(* IEC 61131-3 sources: Elmo_Master/Lasal_PRG/Elmo_EtherCAT_Test_4Axis/Class/LMCControlCommandService (part 3) *)

		groupHeaderPublished := FALSE;
		if restorePreempt & restoredGroupActive then
			// The compact suffix is shared. Restore the complete captured suffix
			// even when the active Group is disjoint from the selected rollback
			// axes, and keep its shared header invalid until every record is done.
			identityHeaderBase := LMC_OWNER_IDENTITY_GROUP_HEADER_BASE;
			OwnershipIdentityState[identityHeaderBase] := 0;
			_memcpy(ptr1:=#OwnershipIdentityState[0],
				ptr2:=#OwnershipPreemptedIdentityState[0],
				cntr:=LMC_OWNER_IDENTITY_SUFFIX_BYTES);
			_memset(dest:=#OwnershipIdentityState[identityHeaderBase],
				usByte:=0, cntr:=40);
			OwnershipIdentityState[identityHeaderBase + 1] :=
				LMC_OWNER_IDENTITY_VERSION;
			OwnershipIdentityState[identityHeaderBase + 2]$UDINT :=
				restoredGroupIdentitySize;
			OwnershipIdentityState[identityHeaderBase + 3]$UDINT :=
				restoredGroupToken;
			OwnershipIdentityState[identityHeaderBase + 4]$UDINT :=
				restoredGroupGeneration;
			OwnershipIdentityState[identityHeaderBase + 5]$UDINT :=
				restoredGroupMask;
			OwnershipIdentityState[identityHeaderBase + 6]$UDINT :=
				restoredGroupSession;
			OwnershipIdentityState[identityHeaderBase + 7]$UDINT :=
				restoredGroupSequence;
			OwnershipIdentityState[identityHeaderBase + 8]$UDINT :=
				TO_UDINT(restoredGroupCommand) or
				(TO_UDINT(restoredGroupReference) shl 16);
			OwnershipIdentityState[identityHeaderBase + 9]$UDINT :=
				TO_UDINT(LMC_OWNER_KIND_GROUP) or
				(TO_UDINT(LMC_OWNER_RESOURCE_AXIS) shl 8) or
				(TO_UDINT(restoredGroupAdmissionMode) shl 16);
			groupHeaderPublished := TRUE;
		end_if;
		axisIndex := 1;
		while axisIndex <= LMC_OWNER_AXIS_COUNT do
			case axisIndex of
				1: axisBit := 0x00000001;
				2: axisBit := 0x00000002;
				3: axisBit := 0x00000004;
				4: axisBit := 0x00000008;
				5: axisBit := 0x00000010;
				6: axisBit := 0x00000020;
				7: axisBit := 0x00000040;
				8: axisBit := 0x00000080;
				9: axisBit := 0x00000100;
			else
				axisBit := 0;
			end_case;
			if (expectedAxisMask and axisBit) <> 0 then
				recordBase := LMC_OWNER_GLOBAL_SLOTS +
					((axisIndex - 1) * LMC_OWNER_AXIS_STRIDE);
				clearIndex := (axisIndex - 1) * LMC_OWNER_AXIS_STRIDE;
				observerBase := (axisIndex - 1) *
					LMC_OWNER_OBSERVER_STRIDE;
				identityHeaderBase := LMC_OWNER_IDENTITY_AXIS_HEADER_BASE +
					((axisIndex - 1) *
					 LMC_OWNER_IDENTITY_AXIS_HEADER_STRIDE);
				OwnershipIdentityState[identityHeaderBase] := 0;
				_memset(dest:=#OwnershipIdentityState[identityHeaderBase],
					usByte:=0,
					cntr:=LMC_OWNER_IDENTITY_AXIS_HEADER_STRIDE * 4);
				if restorePreempt then
					_memcpy(ptr1:=#OwnershipState[recordBase],
						ptr2:=#OwnershipPreemptedState[clearIndex],
						cntr:=LMC_OWNER_AXIS_STRIDE * 4);
					_memcpy(ptr1:=#OwnershipObserverState[observerBase],
						ptr2:=#OwnershipPreemptedIdentityState[
						 LMC_OWNER_PREEMPT_OBSERVER_BASE + observerBase],
						cntr:=LMC_OWNER_OBSERVER_STRIDE * 4);
				else
					_memcpy(ptr1:=#OwnershipState[recordBase],
						ptr2:=#OwnershipLeaseState[clearIndex],
						cntr:=LMC_OWNER_AXIS_STRIDE * 4);
					_memset(dest:=#OwnershipObserverState[observerBase],
						usByte:=0, cntr:=LMC_OWNER_OBSERVER_STRIDE * 4);
				end_if;
				if OwnershipState[recordBase + 1] <> LMC_OWNER_STATE_IDLE then
				identitySize := OwnershipState[recordBase + 15]$UDINT;
				identityTailSize := 0;
				if identitySize > LMC_OWNER_IDENTITY_PREFIX_BYTES then
					identityTailSize := identitySize -
						LMC_OWNER_IDENTITY_PREFIX_BYTES;
				end_if;
				identityPackedCommand :=
					TO_UDINT(OwnershipState[recordBase + 3]) or
					(TO_UDINT(OwnershipState[recordBase + 12]) shl 16);
				identityPackedOwner :=
					TO_UDINT(OwnershipState[recordBase + 2]) or
					(TO_UDINT(OwnershipState[recordBase + 13]) shl 8) or
					(TO_UDINT(OwnershipState[recordBase + 14]) shl 16);
				if OwnershipState[recordBase + 2] =
				   LMC_OWNER_KIND_GROUP then
					if groupHeaderPublished = FALSE then
						identityHeaderBase :=
							LMC_OWNER_IDENTITY_GROUP_HEADER_BASE;
						OwnershipIdentityState[identityHeaderBase] := 0;
						if restorePreempt then
							_memcpy(ptr1:=#OwnershipIdentityState[0],
								ptr2:=#OwnershipPreemptedIdentityState[0],
								cntr:=LMC_OWNER_IDENTITY_SUFFIX_BYTES);
							_memset(dest:=#OwnershipIdentityState[
								identityHeaderBase], usByte:=0, cntr:=40);
							OwnershipIdentityState[identityHeaderBase + 1] :=
								LMC_OWNER_IDENTITY_VERSION;
							OwnershipIdentityState[identityHeaderBase + 2]$UDINT :=
								identitySize;
							OwnershipIdentityState[identityHeaderBase + 3]$UDINT :=
								OwnershipState[recordBase + 4]$UDINT;
							OwnershipIdentityState[identityHeaderBase + 4]$UDINT :=
								OwnershipState[recordBase + 5]$UDINT;
							OwnershipIdentityState[identityHeaderBase + 5]$UDINT :=
								OwnershipState[recordBase + 11]$UDINT;
							OwnershipIdentityState[identityHeaderBase + 6]$UDINT :=
								OwnershipState[recordBase + 6]$UDINT;
							OwnershipIdentityState[identityHeaderBase + 7]$UDINT :=
								OwnershipState[recordBase + 7]$UDINT;
							OwnershipIdentityState[identityHeaderBase + 8]$UDINT :=
								identityPackedCommand;
							OwnershipIdentityState[identityHeaderBase + 9]$UDINT :=
								identityPackedOwner;
						else
							_memcpy(ptr1:=#OwnershipIdentityState[0],
								ptr2:=#OwnershipLeaseIdentityState[0],
								cntr:=LMC_OWNER_IDENTITY_SUFFIX_BYTES);
							_memset(dest:=#OwnershipIdentityState[
								identityHeaderBase], usByte:=0, cntr:=40);
							clearIndex := 1;
							while clearIndex <= 9 do
								OwnershipIdentityState[
									identityHeaderBase + clearIndex] :=
									OwnershipLeaseIdentityState[
									 LMC_OWNER_LEASE_IDENTITY_HEADER_BASE + clearIndex];
								clearIndex += 1;
							end_while;
						end_if;
						groupHeaderPublished := TRUE;
					end_if;
				else
					identityTailOffset :=
						TO_UDINT(OwnershipState[recordBase + 12] - 1) * 8;
					if restorePreempt then
						if identityTailSize > 0 then
							_memset(dest:=#OwnershipIdentityState[
								TO_DINT(identityTailOffset / 4)], usByte:=0,
								cntr:=identityTailSize);
							_memcpy(ptr1:=#OwnershipIdentityState[
								TO_DINT(identityTailOffset / 4)],
								ptr2:=#OwnershipPreemptedIdentityState[
								 TO_DINT(identityTailOffset / 4)],
								cntr:=identityTailSize);
						end_if;
					end_if;
					identityHeaderBase := LMC_OWNER_IDENTITY_AXIS_HEADER_BASE +
						((axisIndex - 1) *
						 LMC_OWNER_IDENTITY_AXIS_HEADER_STRIDE);
					OwnershipIdentityState[identityHeaderBase + 1] :=
						LMC_OWNER_IDENTITY_VERSION;
					OwnershipIdentityState[identityHeaderBase + 2]$UDINT :=
						identitySize;
					OwnershipIdentityState[identityHeaderBase + 3]$UDINT :=
						OwnershipState[recordBase + 4]$UDINT;
					OwnershipIdentityState[identityHeaderBase + 4]$UDINT :=
						OwnershipState[recordBase + 5]$UDINT;
					OwnershipIdentityState[identityHeaderBase + 5]$UDINT :=
						OwnershipState[recordBase + 11]$UDINT;
					OwnershipIdentityState[identityHeaderBase + 6]$UDINT :=
						OwnershipState[recordBase + 6]$UDINT;
					OwnershipIdentityState[identityHeaderBase + 7]$UDINT :=
						OwnershipState[recordBase + 7]$UDINT;
					OwnershipIdentityState[identityHeaderBase + 8]$UDINT :=
						identityPackedCommand;
					OwnershipIdentityState[identityHeaderBase + 9]$UDINT :=
						identityPackedOwner;
					OwnershipIdentityState[identityHeaderBase + 10]$UDINT :=
						identityTailOffset;
					OwnershipIdentityState[identityHeaderBase + 11]$UDINT :=
						identityTailSize;
					OwnershipIdentityState[identityHeaderBase]$UDINT :=
						LMC_OWNER_IDENTITY_AXIS_MAGIC + TO_UDINT(axisIndex);
				end_if;
				end_if;
			end_if;
			axisIndex += 1;
		end_while;
		if groupHeaderPublished then
			OwnershipIdentityState[
				LMC_OWNER_IDENTITY_GROUP_HEADER_BASE]$UDINT :=
				LMC_OWNER_IDENTITY_GROUP_MAGIC;
		end_if;

		if restorePreempt then
			OwnershipPreemptedIdentityState[
				LMC_OWNER_PREEMPT_HEADER_BASE] := 0;
			_memset(dest:=#OwnershipPreemptedState[0], usByte:=0,
				cntr:=sizeof(OwnershipPreemptedState));
			_memset(dest:=#OwnershipPreemptedIdentityState[0], usByte:=0,
				cntr:=sizeof(OwnershipPreemptedIdentityState));
			if restoredGroupActive = FALSE then
				OwnershipLeaseIdentityState[
					LMC_OWNER_LEASE_IDENTITY_HEADER_BASE] := 0;
				_memset(dest:=#OwnershipLeaseState[0], usByte:=0,
					cntr:=sizeof(OwnershipLeaseState));
				_memset(dest:=#OwnershipLeaseIdentityState[0], usByte:=0,
					cntr:=sizeof(OwnershipLeaseIdentityState));
			end_if;
		else
			OwnershipLeaseIdentityState[
				LMC_OWNER_LEASE_IDENTITY_HEADER_BASE] := 0;
			_memset(dest:=#OwnershipLeaseState[0], usByte:=0,
				cntr:=sizeof(OwnershipLeaseState));
			_memset(dest:=#OwnershipLeaseIdentityState[0], usByte:=0,
				cntr:=sizeof(OwnershipLeaseIdentityState));
		end_if;
	elsif Reason = 0 then
		axisIndex := 1;
		while axisIndex <= LMC_OWNER_AXIS_COUNT do
			case axisIndex of
				1: axisBit := 0x00000001;
				2: axisBit := 0x00000002;
				3: axisBit := 0x00000004;
				4: axisBit := 0x00000008;
				5: axisBit := 0x00000010;
				6: axisBit := 0x00000020;
				7: axisBit := 0x00000040;
				8: axisBit := 0x00000080;
				9: axisBit := 0x00000100;
			else
				axisBit := 0;
			end_case;
			if (expectedAxisMask and axisBit) <> 0 then
				recordBase := LMC_OWNER_GLOBAL_SLOTS +
					((axisIndex - 1) * LMC_OWNER_AXIS_STRIDE);
				observerBase := (axisIndex - 1) *
					LMC_OWNER_OBSERVER_STRIDE;
				identityHeaderBase := LMC_OWNER_IDENTITY_AXIS_HEADER_BASE +
					((axisIndex - 1) *
					 LMC_OWNER_IDENTITY_AXIS_HEADER_STRIDE);
				OwnershipIdentityState[identityHeaderBase] := 0;
				_memset(dest:=#OwnershipState[recordBase], usByte:=0,
					cntr:=LMC_OWNER_AXIS_STRIDE * 4);
				OwnershipState[recordBase] := axisIndex;
				OwnershipState[recordBase + 35]$UDINT :=
					LMC_OWNER_AXIS_RECORD_MAGIC + TO_UDINT(axisIndex);
				_memset(dest:=#OwnershipObserverState[observerBase], usByte:=0,
					cntr:=LMC_OWNER_OBSERVER_STRIDE * 4);
			end_if;
			axisIndex += 1;
		end_while;
		if expectedOwnerKind = LMC_OWNER_KIND_GROUP then
			OwnershipIdentityState[
				LMC_OWNER_IDENTITY_GROUP_HEADER_BASE] := 0;
			if expectedAdmissionMode <> LMC_OWNER_ADMISSION_SAFETY then
				_memset(dest:=#OwnershipIdentityState[0], usByte:=0,
					cntr:=LMC_OWNER_IDENTITY_SUFFIX_BYTES);
			end_if;
			_memset(dest:=#OwnershipIdentityState[
				LMC_OWNER_IDENTITY_GROUP_HEADER_BASE], usByte:=0, cntr:=40);
		elsif expectedIdentitySize > LMC_OWNER_IDENTITY_PREFIX_BYTES then
			identityTailSize := expectedIdentitySize -
				LMC_OWNER_IDENTITY_PREFIX_BYTES;
			identityTailOffset := TO_UDINT(expectedReference - 1) * 8;
			_memset(dest:=#OwnershipIdentityState[
				TO_DINT(identityTailOffset / 4)], usByte:=0,
				cntr:=identityTailSize);
		end_if;
	else
		axisIndex := 1;
		while axisIndex <= LMC_OWNER_AXIS_COUNT do
			case axisIndex of
				1: axisBit := 0x00000001;
				2: axisBit := 0x00000002;
				3: axisBit := 0x00000004;
				4: axisBit := 0x00000008;
				5: axisBit := 0x00000010;
				6: axisBit := 0x00000020;
				7: axisBit := 0x00000040;
				8: axisBit := 0x00000080;
				9: axisBit := 0x00000100;
			else
				axisBit := 0;
			end_case;
			if (expectedAxisMask and axisBit) <> 0 then
				recordBase := LMC_OWNER_GLOBAL_SLOTS +
					((axisIndex - 1) * LMC_OWNER_AXIS_STRIDE);
				OwnershipState[recordBase + 1] :=
					LMC_OWNER_STATE_QUARANTINED;
				OwnershipState[recordBase + 32] :=
					LMC_OWNER_REPORT_QUARANTINE;
				OwnershipState[recordBase + 33] := Reason;
			end_if;
			axisIndex += 1;
		end_while;
	end_if;
	if (Reason = 0) &
	   (OwnershipState[7]$UDINT = AdmissionToken) &
	   (OwnershipState[8]$UDINT = OwnerGeneration) then
		OwnershipState[7] := 0;
		OwnershipState[8] := 0;
		OwnershipState[9] := 0;
	end_if;
	if (Reason = 0) &
	   (OwnershipState[10]$UDINT = AdmissionToken) &
	   (OwnershipState[11]$UDINT = OwnerGeneration) then
		OwnershipState[10] := 0;
		OwnershipState[11] := 0;
		OwnershipState[12] := 0;
	end_if;
	if (Reason = 0) &
	   (OwnershipState[13]$UDINT = AdmissionToken) &
	   (OwnershipState[14]$UDINT = OwnerGeneration) then
		OwnershipState[13] := 0;
		OwnershipState[14] := 0;
		OwnershipState[15] := 0;
	end_if;
	Result := 0;

END_FUNCTION

FUNCTION GLOBAL LMCControlCommandService::PublishAxisOwnership
	VAR_INPUT
		AxisMask : UDINT;
		AdmissionToken : UDINT;
		OwnerGeneration : UDINT;
		ReportKind : UINT;
		ReportValue0 : UDINT;
		ReportValue1 : UDINT;
		ObservationCycle : UDINT;
	END_VAR
	VAR_OUTPUT
		Result : DINT;
	END_VAR
	VAR
		axisIndex : DINT;
		axisBit : UDINT;
		recordBase : DINT;
		firstRecordBase : DINT;
		observerBase : DINT;
		observerIndex : DINT;
		identityIndex : DINT;
		clearIndex : DINT;
		identityHeaderBase : DINT;
		identityCompareResult : UDINT;
		expectedResourceKind : DINT;
		expectedOwnerKind : DINT;
		expectedCommandId : DINT;
		expectedAdmissionMode : DINT;
		expectedReference : DINT;
		expectedSession : UDINT;
		expectedSequence : UDINT;
		observerFlags : UDINT;
		identitySize : UDINT;
		identityPrefixSize : UDINT;
		identityTailSize : UDINT;
		identityTailOffset : UDINT;
		identityPackedCommand : UDINT;
		identityPackedOwner : UDINT;
		resourceValid : BOOL;
		selectedFound : BOOL;
		identityShapeValid : BOOL;
		retainGroupLease : BOOL;
		forceQuarantine : BOOL;
		preemptRootValid : BOOL;
		restoreLease : BOOL;
		retainLeaseValid : BOOL;
		destroyBanks : BOOL;
		clearOwner : BOOL;
		groupHeaderPublished : BOOL;
		homeReceiptResult : DINT;
		publishDecisionResult : DINT;
		homeReceiptAxisMaskValid : BOOL;
	END_VAR

	Result := -1;
	if (AxisMask = 0) | (AxisMask > LMC_OWNER_ROBOT_AXIS_MASK) |
	   (AdmissionToken = 0) | (OwnerGeneration = 0) |
	   (ReportKind < LMC_OWNER_REPORT_DISPATCH) |
	   (ReportKind > LMC_OWNER_REPORT_SAFETY_PREEMPT) then
		RETURN;
	end_if;
	homeReceiptResult := HandleAxisOwnershipPublishHomeReceipt(
		AxisMask:=AxisMask, AdmissionToken:=AdmissionToken,
		OwnerGeneration:=OwnerGeneration, ReportKind:=ReportKind,
		ReportValue0:=ReportValue0, ReportValue1:=ReportValue1,
		ObservationCycle:=ObservationCycle);
	if homeReceiptResult <> 2 then
		Result := homeReceiptResult;
		RETURN;
	end_if;
	expectedResourceKind := 0;
	expectedOwnerKind := 0;
	expectedCommandId := 0;
	expectedAdmissionMode := 0;
	expectedReference := 0;
	expectedSession := 0;
	expectedSequence := 0;
	identitySize := 0;
	firstRecordBase := -1;
	selectedFound := FALSE;
	axisIndex := 1;
	while axisIndex <= LMC_OWNER_AXIS_COUNT do
		case axisIndex of
			1: axisBit := 0x00000001;
			2: axisBit := 0x00000002;
			3: axisBit := 0x00000004;
			4: axisBit := 0x00000008;
			5: axisBit := 0x00000010;
			6: axisBit := 0x00000020;
			7: axisBit := 0x00000040;
			8: axisBit := 0x00000080;
			9: axisBit := 0x00000100;
		else
			axisBit := 0;
		end_case;
		recordBase := LMC_OWNER_GLOBAL_SLOTS +
			((axisIndex - 1) * LMC_OWNER_AXIS_STRIDE);
		if (AxisMask and axisBit) <> 0 then
			if selectedFound = FALSE then
				expectedResourceKind := OwnershipState[recordBase + 13];
				expectedOwnerKind := OwnershipState[recordBase + 2];
				expectedCommandId := OwnershipState[recordBase + 3];
				expectedAdmissionMode := OwnershipState[recordBase + 14];
				expectedReference := OwnershipState[recordBase + 12];
				expectedSession := OwnershipState[recordBase + 6]$UDINT;
				expectedSequence := OwnershipState[recordBase + 7]$UDINT;
				identitySize := OwnershipState[recordBase + 15]$UDINT;
				firstRecordBase := recordBase;
				selectedFound := TRUE;
			end_if;
			if (OwnershipState[recordBase] <> axisIndex) |
			   (OwnershipState[recordBase + 35]$UDINT <>
			    (LMC_OWNER_AXIS_RECORD_MAGIC + TO_UDINT(axisIndex))) |
			   (OwnershipState[recordBase + 4]$UDINT <>
			    AdmissionToken) |
			   (OwnershipState[recordBase + 5]$UDINT <>
			    OwnerGeneration) |
			   (OwnershipState[recordBase + 11]$UDINT <> AxisMask) |
			   (OwnershipState[recordBase + 13] <>
			    expectedResourceKind) |
			   (OwnershipState[recordBase + 2] <> expectedOwnerKind) |
			   (OwnershipState[recordBase + 3] <> expectedCommandId) |
			   (OwnershipState[recordBase + 14] <>
			    expectedAdmissionMode) |
			   (OwnershipState[recordBase + 12] <>
			    expectedReference) |
			   (OwnershipState[recordBase + 6]$UDINT <> expectedSession) |
			   (OwnershipState[recordBase + 7]$UDINT <> expectedSequence) |
			   (OwnershipState[recordBase + 15]$UDINT <> identitySize) then
				Result := -2;
				RETURN;
			elsif (OwnershipState[recordBase + 1] =
			       LMC_OWNER_STATE_QUARANTINED) &
			      (ReportKind <> LMC_OWNER_REPORT_QUARANTINE) then
				Result := -3;
				RETURN;
			end_if;
		elsif (OwnershipState[recordBase + 4]$UDINT = AdmissionToken) |
		      (OwnershipState[recordBase + 5]$UDINT = OwnerGeneration) then
			Result := -2;
			RETURN;
		end_if;
		axisIndex += 1;
	end_while;
	if selectedFound = FALSE then
		Result := -2;
		RETURN;
	end_if;
	identityShapeValid := FALSE;
	if expectedCommandId = 0x2023 then
		identityShapeValid := identitySize = 8;
	elsif expectedCommandId = 0x2024 then
		identityShapeValid := identitySize = 1;
	elsif expectedCommandId = 0x2022 then
		identityShapeValid := identitySize = 16;
	elsif (expectedCommandId = 0x209F) | (expectedCommandId = 0x20A0) then
		identityShapeValid := identitySize = 32;
	elsif expectedCommandId = 0x20A2 then
		identityShapeValid := identitySize = 24;
	elsif (expectedCommandId = 0x2047) | (expectedCommandId = 0x2048) |
	      (expectedCommandId = 0x2049) | (expectedCommandId = 0x204A) |
	      (expectedCommandId = 0x204B) then
		identityShapeValid := identitySize = 1;
	elsif expectedCommandId = 0x2085 then
		identityShapeValid := identitySize = 16;
	elsif expectedCommandId = 0x20A4 then
		identityShapeValid := identitySize = 96;
	elsif expectedCommandId = 0x7D22 then
		identityShapeValid := identitySize = 104;
	elsif expectedCommandId = 0x20E7 then
		identityShapeValid := identitySize = 1320;
	elsif expectedCommandId = 0x7D13 then
		identityShapeValid := identitySize = 56;
	elsif (expectedCommandId = 0x7D15) |
	      (expectedCommandId = 0x7E53) then
		identityShapeValid := identitySize = 72;
	end_if;
	identityPrefixSize := identitySize;
	if identityPrefixSize > LMC_OWNER_IDENTITY_PREFIX_BYTES then
		identityPrefixSize := LMC_OWNER_IDENTITY_PREFIX_BYTES;
	end_if;
	identityTailSize := 0;
	if identitySize > LMC_OWNER_IDENTITY_PREFIX_BYTES then
		identityTailSize := identitySize - LMC_OWNER_IDENTITY_PREFIX_BYTES;
	end_if;
	identityTailOffset := 0;
	if expectedOwnerKind <> LMC_OWNER_KIND_GROUP then
		if (expectedReference < 1) |
		   (expectedReference > LMC_OWNER_AXIS_COUNT) then
			identityShapeValid := FALSE;
		else
			identityTailOffset := TO_UDINT(expectedReference - 1) * 8;
		end_if;
		if identityTailSize > 8 then
			identityShapeValid := FALSE;
		end_if;
	end_if;
	if (identityTailOffset + identityTailSize) >
	   LMC_OWNER_IDENTITY_SUFFIX_BYTES then
		identityShapeValid := FALSE;
	end_if;
	identityPackedCommand := TO_UDINT(expectedCommandId) or
		(TO_UDINT(expectedReference) shl 16);
	identityPackedOwner := TO_UDINT(expectedOwnerKind) or
		(TO_UDINT(expectedResourceKind) shl 8) or
		(TO_UDINT(expectedAdmissionMode) shl 16);
	axisIndex := 1;
	while axisIndex <= LMC_OWNER_AXIS_COUNT do
		case axisIndex of
			1: axisBit := 0x00000001;
			2: axisBit := 0x00000002;
			3: axisBit := 0x00000004;
			4: axisBit := 0x00000008;
			5: axisBit := 0x00000010;
			6: axisBit := 0x00000020;
			7: axisBit := 0x00000040;
			8: axisBit := 0x00000080;
			9: axisBit := 0x00000100;
		else
			axisBit := 0;
		end_case;
		if (AxisMask and axisBit) <> 0 then
			recordBase := LMC_OWNER_GLOBAL_SLOTS +
				((axisIndex - 1) * LMC_OWNER_AXIS_STRIDE);
			if expectedOwnerKind = LMC_OWNER_KIND_GROUP then
				identityHeaderBase := LMC_OWNER_IDENTITY_GROUP_HEADER_BASE;
				if (OwnershipIdentityState[identityHeaderBase]$UDINT <>
				    LMC_OWNER_IDENTITY_GROUP_MAGIC) |
				   (OwnershipIdentityState[identityHeaderBase + 1] <>
				    LMC_OWNER_IDENTITY_VERSION) |
				   (OwnershipIdentityState[identityHeaderBase + 2]$UDINT <>
				    identitySize) |
				   (OwnershipIdentityState[identityHeaderBase + 3]$UDINT <>
				    AdmissionToken) |
				   (OwnershipIdentityState[identityHeaderBase + 4]$UDINT <>
				    OwnerGeneration) |
				   (OwnershipIdentityState[identityHeaderBase + 5]$UDINT <>
				    AxisMask) |
				   (OwnershipIdentityState[identityHeaderBase + 6]$UDINT <>
				    expectedSession) |
				   (OwnershipIdentityState[identityHeaderBase + 7]$UDINT <>
				    expectedSequence) |
				   (OwnershipIdentityState[identityHeaderBase + 8]$UDINT <>
				    identityPackedCommand) |
				   (OwnershipIdentityState[identityHeaderBase + 9]$UDINT <>
				    identityPackedOwner) then
					identityShapeValid := FALSE;
				end_if;
			else
				identityHeaderBase := LMC_OWNER_IDENTITY_AXIS_HEADER_BASE +
					((axisIndex - 1) * LMC_OWNER_IDENTITY_AXIS_HEADER_STRIDE);
				if (OwnershipIdentityState[identityHeaderBase]$UDINT <>
				    (LMC_OWNER_IDENTITY_AXIS_MAGIC + TO_UDINT(axisIndex))) |
				   (OwnershipIdentityState[identityHeaderBase + 1] <>
				    LMC_OWNER_IDENTITY_VERSION) |
				   (OwnershipIdentityState[identityHeaderBase + 2]$UDINT <>
				    identitySize) |
				   (OwnershipIdentityState[identityHeaderBase + 3]$UDINT <>
				    AdmissionToken) |
				   (OwnershipIdentityState[identityHeaderBase + 4]$UDINT <>
				    OwnerGeneration) |
				   (OwnershipIdentityState[identityHeaderBase + 5]$UDINT <>
				    AxisMask) |
				   (OwnershipIdentityState[identityHeaderBase + 6]$UDINT <>
				    expectedSession) |
				   (OwnershipIdentityState[identityHeaderBase + 7]$UDINT <>
				    expectedSequence) |
				   (OwnershipIdentityState[identityHeaderBase + 8]$UDINT <>
				    identityPackedCommand) |
				   (OwnershipIdentityState[identityHeaderBase + 9]$UDINT <>
				    identityPackedOwner) |
				   (OwnershipIdentityState[identityHeaderBase + 10]$UDINT <>
				    identityTailOffset) |
				   (OwnershipIdentityState[identityHeaderBase + 11]$UDINT <>
				    identityTailSize) then
					identityShapeValid := FALSE;
				end_if;
			end_if;
			identityCompareResult := _memcmp(
				ptr1:=#OwnershipState[firstRecordBase + 16],
				ptr2:=#OwnershipState[recordBase + 16],
				cntr:=identityPrefixSize);
			if identityCompareResult <> 0 then
				identityShapeValid := FALSE;
			end_if;
		end_if;
		axisIndex += 1;
	end_while;
	if identityShapeValid = FALSE then
		OwnershipState[24] := 1;
		Result := -3;
		RETURN;
	end_if;
	resourceValid := FALSE;
	case expectedResourceKind of
		LMC_OWNER_RESOURCE_AXIS:
			resourceValid :=
				(OwnershipState[7]$UDINT <> AdmissionToken) &
				(OwnershipState[8]$UDINT <> OwnerGeneration) &
				(OwnershipState[10]$UDINT <> AdmissionToken) &
				(OwnershipState[11]$UDINT <> OwnerGeneration) &
				(OwnershipState[13]$UDINT <> AdmissionToken) &
				(OwnershipState[14]$UDINT <> OwnerGeneration);
		LMC_OWNER_RESOURCE_LMC_HOME_ENGINE:
			resourceValid :=
				(OwnershipState[7]$UDINT = AdmissionToken) &
				(OwnershipState[8]$UDINT = OwnerGeneration) &
				(OwnershipState[9]$UDINT = AxisMask) &
				(OwnershipState[10]$UDINT <> AdmissionToken) &
				(OwnershipState[11]$UDINT <> OwnerGeneration) &
				(OwnershipState[13]$UDINT <> AdmissionToken) &
				(OwnershipState[14]$UDINT <> OwnerGeneration);
		LMC_OWNER_RESOURCE_DS402_HOME_ENGINE:
			resourceValid :=
				(OwnershipState[10]$UDINT = AdmissionToken) &
				(OwnershipState[11]$UDINT = OwnerGeneration) &
				(OwnershipState[12]$UDINT = AxisMask) &
				(OwnershipState[7]$UDINT <> AdmissionToken) &
				(OwnershipState[8]$UDINT <> OwnerGeneration) &
				(OwnershipState[13]$UDINT <> AdmissionToken) &
				(OwnershipState[14]$UDINT <> OwnerGeneration);
		LMC_OWNER_RESOURCE_DIAGNOSTICS_SDO_ENGINE:
			resourceValid :=
				(OwnershipState[13]$UDINT = AdmissionToken) &
				(OwnershipState[14]$UDINT = OwnerGeneration) &
				(OwnershipState[15]$UDINT = AxisMask) &
				(OwnershipState[7]$UDINT <> AdmissionToken) &
				(OwnershipState[8]$UDINT <> OwnerGeneration) &
				(OwnershipState[10]$UDINT <> AdmissionToken) &
				(OwnershipState[11]$UDINT <> OwnerGeneration);
	else
	end_case;
	if resourceValid = FALSE then
		Result := -2;
		RETURN;
	end_if;

	publishDecisionResult := PrepareAxisOwnershipPublishDecision(
		AxisMask:=AxisMask, AdmissionToken:=AdmissionToken,
		OwnerGeneration:=OwnerGeneration, ReportKind:=ReportKind,
		ExpectedSession:=expectedSession,
		ExpectedSequence:=expectedSequence,
		ExpectedCommandId:=expectedCommandId,
		ExpectedReference:=expectedReference,
		ExpectedAdmissionMode:=expectedAdmissionMode,
		ExpectedOwnerKind:=expectedOwnerKind);
	if publishDecisionResult < 0 then
		Result := publishDecisionResult;
		RETURN;
	elsif publishDecisionResult > 7 then
		Result := -3;
		RETURN;
	end_if;
	preemptRootValid := (publishDecisionResult and 1) <> 0;
	forceQuarantine := (publishDecisionResult and 2) <> 0;
	restoreLease := (publishDecisionResult and 4) <> 0;
	destroyBanks :=
		(ReportKind = LMC_OWNER_REPORT_TERMINAL_SUCCESS) &
		((expectedCommandId = 0x2048) | (expectedCommandId = 0x204B));
	retainGroupLease :=
		(ReportKind = LMC_OWNER_REPORT_TERMINAL_SUCCESS) &
		(forceQuarantine = FALSE) &
		(expectedOwnerKind = LMC_OWNER_KIND_GROUP) &
		(expectedCommandId = 0x2047);
	if retainGroupLease then
		// A successful GroupEnable establishes its own accepted exact lease;
		// it does not restore or synthesize a prior lease record.
		retainLeaseValid :=
			(expectedResourceKind = LMC_OWNER_RESOURCE_AXIS) &
			(expectedAdmissionMode = LMC_OWNER_ADMISSION_ORDINARY) &
			(expectedReference = 0x0100) &
			(AxisMask = LMC_OWNER_PROFILE_AXIS_MASK) &
			(expectedSession <> 0) & (expectedSequence <> 0) &
			(identitySize = 1) &
			(OwnershipIdentityState[
			 LMC_OWNER_IDENTITY_GROUP_HEADER_BASE]$UDINT =
			 LMC_OWNER_IDENTITY_GROUP_MAGIC) &
			(OwnershipIdentityState[
			 LMC_OWNER_IDENTITY_GROUP_HEADER_BASE + 1] =
			 LMC_OWNER_IDENTITY_VERSION) &
			(OwnershipIdentityState[
			 LMC_OWNER_IDENTITY_GROUP_HEADER_BASE + 2]$UDINT = 1) &
			(OwnershipIdentityState[
			 LMC_OWNER_IDENTITY_GROUP_HEADER_BASE + 3]$UDINT =
			 AdmissionToken) &
			(OwnershipIdentityState[
			 LMC_OWNER_IDENTITY_GROUP_HEADER_BASE + 4]$UDINT =
			 OwnerGeneration) &
			(OwnershipIdentityState[
			 LMC_OWNER_IDENTITY_GROUP_HEADER_BASE + 5]$UDINT = AxisMask) &
			(OwnershipIdentityState[
			 LMC_OWNER_IDENTITY_GROUP_HEADER_BASE + 6]$UDINT =
			 expectedSession) &
			(OwnershipIdentityState[
			 LMC_OWNER_IDENTITY_GROUP_HEADER_BASE + 7]$UDINT =
			 expectedSequence) &
			(OwnershipIdentityState[
			 LMC_OWNER_IDENTITY_GROUP_HEADER_BASE + 8]$UDINT =
			 (TO_UDINT(0x2047) or (TO_UDINT(0x0100) shl 16))) &
			(OwnershipIdentityState[
			 LMC_OWNER_IDENTITY_GROUP_HEADER_BASE + 9]$UDINT =
			 (TO_UDINT(LMC_OWNER_KIND_GROUP) or
			  (TO_UDINT(LMC_OWNER_RESOURCE_AXIS) shl 8) or
			  (TO_UDINT(LMC_OWNER_ADMISSION_ORDINARY) shl 16)));
		axisIndex := 1;
		while axisIndex <= LMC_OWNER_AXIS_COUNT do
			case axisIndex of
				1: axisBit := 0x00000001;
				2: axisBit := 0x00000002;
				3: axisBit := 0x00000004;
				4: axisBit := 0x00000008;
				5: axisBit := 0x00000010;
				6: axisBit := 0x00000020;
				7: axisBit := 0x00000040;
				8: axisBit := 0x00000080;
				9: axisBit := 0x00000100;
			else
				axisBit := 0;
			end_case;
			if (AxisMask and axisBit) <> 0 then
				recordBase := LMC_OWNER_GLOBAL_SLOTS +
					((axisIndex - 1) * LMC_OWNER_AXIS_STRIDE);
				if OwnershipState[recordBase + 16]$UDINT <> 1 then
					retainLeaseValid := FALSE;
				end_if;
				identityIndex := 17;
				while identityIndex <= 31 do
					if OwnershipState[recordBase + identityIndex] <> 0 then
						retainLeaseValid := FALSE;
					end_if;
					identityIndex += 1;
				end_while;
				identityCompareResult := _memcmp(
					ptr1:=#OwnershipState[firstRecordBase + 16],
					ptr2:=#OwnershipState[recordBase + 16], cntr:=1);
				if identityCompareResult <> 0 then
					retainLeaseValid := FALSE;
				end_if;
			end_if;
			axisIndex += 1;
		end_while;
		identityIndex := 0;
		while identityIndex < LMC_OWNER_IDENTITY_SUFFIX_DINTS do
			if OwnershipIdentityState[identityIndex] <> 0 then
				retainLeaseValid := FALSE;
			end_if;
			identityIndex += 1;
		end_while;
		if retainLeaseValid = FALSE then
			OwnershipState[24] := 1;
			Result := -3;
			RETURN;
		end_if;
	end_if;
	clearOwner :=
		(ReportKind = LMC_OWNER_REPORT_TERMINAL_SUCCESS) &
		(forceQuarantine = FALSE) &
		(restoreLease = FALSE) & (retainGroupLease = FALSE);
	if ReportKind = LMC_OWNER_REPORT_TERMINAL_SAFE_FAILURE then
		clearOwner := (expectedOwnerKind <> LMC_OWNER_KIND_DIRECT) &
			(expectedOwnerKind <> LMC_OWNER_KIND_GROUP) &
			(forceQuarantine = FALSE);
	end_if;
	if (expectedCommandId = 0x7D13) &
	   (expectedOwnerKind = LMC_OWNER_KIND_LMC_HOME) &
	   (expectedResourceKind = LMC_OWNER_RESOURCE_LMC_HOME_ENGINE) &
	   (expectedAdmissionMode = LMC_OWNER_ADMISSION_LIFECYCLE) &
	   (preemptRootValid = FALSE) & (forceQuarantine = FALSE) &
	   clearOwner &
	   ((ReportKind = LMC_OWNER_REPORT_TERMINAL_SUCCESS) |
	    (ReportKind = LMC_OWNER_REPORT_TERMINAL_SAFE_FAILURE)) then
		// Publish an immutable exact receipt before any owner surface is cleared.
		// The caller accepts the receipt and replays this call to perform cleanup.
		homeReceiptAxisMaskValid := FALSE;
		case expectedReference of
			1: homeReceiptAxisMaskValid := AxisMask = 0x00000001;
			2: homeReceiptAxisMaskValid := AxisMask = 0x00000002;
			3: homeReceiptAxisMaskValid := AxisMask = 0x00000004;
			4: homeReceiptAxisMaskValid := AxisMask = 0x00000008;
		else
		end_case;
		if (homeReceiptAxisMaskValid = FALSE) |
		   (ZeroHomeState[51]$UDINT <> LMC_HOME_RECORD_MAGIC) |
		   (ZeroHomeState[33]$UDINT = 0) |
		   (ZeroHomeState[34]$UDINT <> AdmissionToken) |
		   (ZeroHomeState[35]$UDINT <> OwnerGeneration) |
		   (ZeroHomeState[36]$UDINT <> expectedSession) |
		   (ZeroHomeState[37]$UDINT <> expectedSequence) |
		   (ZeroHomeState[38]$UDINT <> AxisMask) |
		   (ZeroHomeState[39] <> LMC_HOME_ENGINE_FINALIZE) |
		   (ZeroHomeState[57]$UDINT <> ReportValue0) |
		   (ZeroHomeState[58] <> TO_DINT(ReportKind)) |
		   (ZeroHomeState[59] <> 0) |
		   (ZeroHomeState[31]$UDINT <> ReportValue1) |
		   (ZeroHomeState[46]$UDINT <> ObservationCycle) |
		   ((ZeroHomeState[56]$UDINT and
		     LMC_HOME_FLAG_OWNER_FINALIZE_INTENT) = 0) |
		   ((ZeroHomeState[56]$UDINT and
		     LMC_HOME_FLAG_OWNER_FINALIZE_ACCEPTED) <> 0) |
		   (ZeroHomeState[60] <> 0) then
			OwnershipState[24] := 1;
			Result := -3;
			RETURN;
		end_if;
		ZeroHomeState[60] := 0;
		ZeroHomeState[61] := LMC_HOME_OWNER_RECEIPT_PREPARED;
		ZeroHomeState[62] := 0;
		ZeroHomeState[63]$UDINT := ZeroHomeState[33]$UDINT;
		ZeroHomeState[60]$UDINT := LMC_HOME_OWNER_RECEIPT_MAGIC;
		Result := 0;
		RETURN;
	end_if;
	axisIndex := 1;
	while axisIndex <= LMC_OWNER_AXIS_COUNT do
		case axisIndex of
			1: axisBit := 0x00000001;
			2: axisBit := 0x00000002;
			3: axisBit := 0x00000004;
			4: axisBit := 0x00000008;
			5: axisBit := 0x00000010;
			6: axisBit := 0x00000020;
			7: axisBit := 0x00000040;
			8: axisBit := 0x00000080;
			9: axisBit := 0x00000100;
		else
			axisBit := 0;
		end_case;
		if (AxisMask and axisBit) <> 0 then
			recordBase := LMC_OWNER_GLOBAL_SLOTS +
				((axisIndex - 1) * LMC_OWNER_AXIS_STRIDE);
			observerBase := (axisIndex - 1) * LMC_OWNER_OBSERVER_STRIDE;
			OwnershipState[recordBase + 9]$UDINT := ObservationCycle;
			OwnershipState[recordBase + 32] := TO_DINT(ReportKind);
			OwnershipState[recordBase + 33]$UDINT := ReportValue0;
			OwnershipState[recordBase + 34]$UDINT := ReportValue1;
			case ReportKind of
				LMC_OWNER_REPORT_TERMINAL_SUCCESS:
					if forceQuarantine then
						OwnershipState[recordBase + 1] :=
							LMC_OWNER_STATE_QUARANTINED;
						OwnershipState[recordBase + 32] :=
							LMC_OWNER_REPORT_QUARANTINE;
					elsif restoreLease then
						// Exact lease restore is applied after this validation loop.
					elsif retainGroupLease then
						OwnershipState[recordBase + 1] :=
							LMC_OWNER_STATE_GROUP_LEASE;
						observerIndex := 0;
						while observerIndex < LMC_OWNER_OBSERVER_STRIDE do
							OwnershipObserverState[observerBase + observerIndex] := 0;
							observerIndex += 1;
						end_while;
					elsif clearOwner then
						_memset(dest:=#OwnershipState[recordBase], usByte:=0,
							cntr:=LMC_OWNER_AXIS_STRIDE * 4);
						OwnershipState[recordBase] := axisIndex;
						OwnershipState[recordBase + 35]$UDINT :=
							LMC_OWNER_AXIS_RECORD_MAGIC + TO_UDINT(axisIndex);
						_memset(dest:=#OwnershipObserverState[observerBase],
							usByte:=0, cntr:=LMC_OWNER_OBSERVER_STRIDE * 4);
					end_if;
				LMC_OWNER_REPORT_TERMINAL_SAFE_FAILURE:
					if (expectedOwnerKind = LMC_OWNER_KIND_DIRECT) |
					   (expectedOwnerKind = LMC_OWNER_KIND_GROUP) |
					   forceQuarantine then
						OwnershipState[recordBase + 1] :=
							LMC_OWNER_STATE_QUARANTINED;
					elsif clearOwner then
						_memset(dest:=#OwnershipState[recordBase], usByte:=0,
							cntr:=LMC_OWNER_AXIS_STRIDE * 4);
						OwnershipState[recordBase] := axisIndex;
						OwnershipState[recordBase + 35]$UDINT :=
							LMC_OWNER_AXIS_RECORD_MAGIC + TO_UDINT(axisIndex);
						_memset(dest:=#OwnershipObserverState[observerBase],
							usByte:=0, cntr:=LMC_OWNER_OBSERVER_STRIDE * 4);
					end_if;
				LMC_OWNER_REPORT_QUARANTINE:
					OwnershipState[recordBase + 1] :=
						LMC_OWNER_STATE_QUARANTINED;
				LMC_OWNER_REPORT_SAFETY_PREEMPT:
					OwnershipState[recordBase + 1] :=
						LMC_OWNER_STATE_SAFETY_PREEMPTING;
			else
			end_case;
		end_if;
		axisIndex += 1;
	end_while;

	if restoreLease then
		OwnershipIdentityState[
			LMC_OWNER_IDENTITY_GROUP_HEADER_BASE] := 0;
		_memcpy(ptr1:=#OwnershipIdentityState[0],
			ptr2:=#OwnershipLeaseIdentityState[0],
			cntr:=LMC_OWNER_IDENTITY_SUFFIX_BYTES);
		_memset(dest:=#OwnershipIdentityState[
			LMC_OWNER_IDENTITY_GROUP_HEADER_BASE], usByte:=0, cntr:=40);
		clearIndex := 1;
		while clearIndex <= 9 do
			OwnershipIdentityState[
				LMC_OWNER_IDENTITY_GROUP_HEADER_BASE + clearIndex] :=
				OwnershipLeaseIdentityState[
				 LMC_OWNER_LEASE_IDENTITY_HEADER_BASE + clearIndex];
			clearIndex += 1;
		end_while;
		axisIndex := 1;
		while axisIndex <= LMC_OWNER_AXIS_COUNT do
			case axisIndex of
				1: axisBit := 0x00000001;
				2: axisBit := 0x00000002;
				3: axisBit := 0x00000004;
				4: axisBit := 0x00000008;
				5: axisBit := 0x00000010;
				6: axisBit := 0x00000020;
				7: axisBit := 0x00000040;
				8: axisBit := 0x00000080;
				9: axisBit := 0x00000100;
			else
				axisBit := 0;
			end_case;
			if (AxisMask and axisBit) <> 0 then
				recordBase := LMC_OWNER_GLOBAL_SLOTS +
					((axisIndex - 1) * LMC_OWNER_AXIS_STRIDE);
				clearIndex := (axisIndex - 1) * LMC_OWNER_AXIS_STRIDE;
				observerBase := (axisIndex - 1) *
					LMC_OWNER_OBSERVER_STRIDE;
				identityTailOffset := LMC_OWNER_IDENTITY_AXIS_HEADER_BASE +
					TO_UDINT((axisIndex - 1) *
					 LMC_OWNER_IDENTITY_AXIS_HEADER_STRIDE);
				OwnershipIdentityState[TO_DINT(identityTailOffset)] := 0;
				_memset(dest:=#OwnershipIdentityState[
					TO_DINT(identityTailOffset)], usByte:=0,
					cntr:=LMC_OWNER_IDENTITY_AXIS_HEADER_STRIDE * 4);
				_memcpy(ptr1:=#OwnershipState[recordBase],
					ptr2:=#OwnershipLeaseState[clearIndex],
					cntr:=LMC_OWNER_AXIS_STRIDE * 4);
				_memset(dest:=#OwnershipObserverState[observerBase], usByte:=0,
					cntr:=LMC_OWNER_OBSERVER_STRIDE * 4);
			end_if;
			axisIndex += 1;
		end_while;
		OwnershipIdentityState[
			LMC_OWNER_IDENTITY_GROUP_HEADER_BASE]$UDINT :=
			LMC_OWNER_IDENTITY_GROUP_MAGIC;
	end_if;

	if clearOwner then
		axisIndex := 1;
		while axisIndex <= LMC_OWNER_AXIS_COUNT do
			case axisIndex of
				1: axisBit := 0x00000001;
				2: axisBit := 0x00000002;
				3: axisBit := 0x00000004;
				4: axisBit := 0x00000008;
				5: axisBit := 0x00000010;
				6: axisBit := 0x00000020;
				7: axisBit := 0x00000040;
				8: axisBit := 0x00000080;
				9: axisBit := 0x00000100;
			else
				axisBit := 0;
			end_case;
			if (AxisMask and axisBit) <> 0 then
				identityTailOffset := LMC_OWNER_IDENTITY_AXIS_HEADER_BASE +
					TO_UDINT((axisIndex - 1) *
					 LMC_OWNER_IDENTITY_AXIS_HEADER_STRIDE);
				_memset(dest:=#OwnershipIdentityState[
					TO_DINT(identityTailOffset)], usByte:=0,
					cntr:=LMC_OWNER_IDENTITY_AXIS_HEADER_STRIDE * 4);
			end_if;
			axisIndex += 1;
		end_while;
		if expectedOwnerKind = LMC_OWNER_KIND_GROUP then
			OwnershipIdentityState[
				LMC_OWNER_IDENTITY_GROUP_HEADER_BASE] := 0;
			if expectedAdmissionMode <> LMC_OWNER_ADMISSION_SAFETY then
				_memset(dest:=#OwnershipIdentityState[0], usByte:=0,
					cntr:=LMC_OWNER_IDENTITY_SUFFIX_BYTES);
			end_if;
			_memset(dest:=#OwnershipIdentityState[
				LMC_OWNER_IDENTITY_GROUP_HEADER_BASE], usByte:=0, cntr:=40);
		elsif identityTailSize > 0 then
			identityTailOffset := TO_UDINT(expectedReference - 1) * 8;
			_memset(dest:=#OwnershipIdentityState[
				TO_DINT(identityTailOffset / 4)], usByte:=0,
				cntr:=identityTailSize);
		end_if;
	end_if;

	if (ReportKind = LMC_OWNER_REPORT_TERMINAL_SUCCESS) &
	   (forceQuarantine = FALSE) then
		if preemptRootValid then
			OwnershipPreemptedIdentityState[
				LMC_OWNER_PREEMPT_HEADER_BASE] := 0;
			_memset(dest:=#OwnershipPreemptedState[0], usByte:=0,
				cntr:=sizeof(OwnershipPreemptedState));
			_memset(dest:=#OwnershipPreemptedIdentityState[0], usByte:=0,
				cntr:=sizeof(OwnershipPreemptedIdentityState));
		end_if;
		if restoreLease | destroyBanks then
			OwnershipLeaseIdentityState[
				LMC_OWNER_LEASE_IDENTITY_HEADER_BASE] := 0;
			_memset(dest:=#OwnershipLeaseState[0], usByte:=0,
				cntr:=sizeof(OwnershipLeaseState));
			_memset(dest:=#OwnershipLeaseIdentityState[0], usByte:=0,
				cntr:=sizeof(OwnershipLeaseIdentityState));
		end_if;
	end_if;

	if (ReportKind = LMC_OWNER_REPORT_TERMINAL_SUCCESS) |
	   (ReportKind = LMC_OWNER_REPORT_TERMINAL_SAFE_FAILURE) then
		if (OwnershipState[7]$UDINT = AdmissionToken) &
		   (OwnershipState[8]$UDINT = OwnerGeneration) then
			OwnershipState[7] := 0;
			OwnershipState[8] := 0;
			OwnershipState[9] := 0;
		end_if;
		if (OwnershipState[10]$UDINT = AdmissionToken) &
		   (OwnershipState[11]$UDINT = OwnerGeneration) then
			OwnershipState[10] := 0;
			OwnershipState[11] := 0;
			OwnershipState[12] := 0;
		end_if;
		if (OwnershipState[13]$UDINT = AdmissionToken) &
		   (OwnershipState[14]$UDINT = OwnerGeneration) then
			OwnershipState[13] := 0;
			OwnershipState[14] := 0;
			OwnershipState[15] := 0;
		end_if;
	end_if;
	Result := 0;

END_FUNCTION

FUNCTION GLOBAL LMCControlCommandService::ReconcileAxisOwnershipStartup
	VAR_INPUT
		DiagnosticsBootId 	: UDINT;
		ObservationCycle 	: UDINT;
		ReportCycle 	: UDINT;
		DiagnosticsDrainFlags 	: UDINT;
	END_VAR
	VAR_OUTPUT
		Result 	: DINT;
	END_VAR
	VAR
		startupSnapshot : ARRAY [0..11] OF UDINT;
		copyResult : DINT;
		axisIndex : DINT;
		recordBase : DINT;
		stateIndex : DINT;
		combinedProof : UDINT;
		groupSignature : UDINT;
		robotState : DINT;
		profileLockState : DINT;
		profileFinished : DINT;
		stableElapsedMilliseconds : UDINT;
		tableIdle : BOOL;
		physicalIdle : BOOL;
		groupIdle : BOOL;
		drained : BOOL;
		signatureStable : BOOL;
		freshObservation : BOOL;
		auxiliaryIdle : BOOL;
	END_VAR

	Result := -1;
	if (DiagnosticsBootId = 0) | (ObservationCycle = 0) |
		(ReportCycle = 0) then
		RETURN;
	end_if;

	// Normal operations may make a completed same-boot table non-idle. Do not
	// reinterpret those transient states as startup failures.
	if (OwnershipState[0]$UDINT = LMC_OWNER_TABLE_MAGIC) &
		(OwnershipState[3]$UDINT = DiagnosticsBootId) then
		if (OwnershipState[4]$UDINT <> 0) &
			(OwnershipState[5]$UDINT = LMC_OWNER_STARTUP_PROOF_REQUIRED) &
			(OwnershipState[6] = 0) &
			(OwnershipState[24] = 0) then
			Result := 0;
		else
			Result := -3;
		end_if;
		RETURN;
	end_if;

	auxiliaryIdle := TRUE;
	stateIndex := 0;
	while stateIndex <= 431 do
		if (OwnershipIdentityState[stateIndex] <> 0) |
		   (OwnershipPreemptedIdentityState[stateIndex] <> 0) then
			auxiliaryIdle := FALSE;
		end_if;
		stateIndex += 1;
	end_while;
	stateIndex := 0;
	while stateIndex <= 323 do
		if (OwnershipLeaseState[stateIndex] <> 0) |
		   (OwnershipPreemptedState[stateIndex] <> 0) |
		   (OwnershipLeaseIdentityState[stateIndex] <> 0) then
			auxiliaryIdle := FALSE;
		end_if;
		stateIndex += 1;
	end_while;
	if auxiliaryIdle = FALSE then
		Result := -3;
		RETURN;
	end_if;

	// A nonzero existing table may be replaced only when it is a valid,
	// prior-boot, completely idle owner table.
	if OwnershipState[0]$UDINT = 0 then
		tableIdle := TRUE;
		stateIndex := 1;
		while stateIndex <= 351 do
			if OwnershipState[stateIndex] <> 0 then
				tableIdle := FALSE;
			end_if;
			stateIndex += 1;
		end_while;
		if tableIdle = FALSE then
			Result := -3;
			RETURN;
		end_if;
	elsif OwnershipState[0]$UDINT = LMC_OWNER_TABLE_MAGIC then
		tableIdle := (OwnershipState[3]$UDINT <> 0) &
			(OwnershipState[4]$UDINT <> 0) &
			(OwnershipState[5]$UDINT = LMC_OWNER_STARTUP_PROOF_REQUIRED) &
			(OwnershipState[6] = 0) &
			(OwnershipState[7] = 0) & (OwnershipState[8] = 0) &
			(OwnershipState[9] = 0) & (OwnershipState[10] = 0) &
			(OwnershipState[11] = 0) & (OwnershipState[12] = 0) &
			(OwnershipState[13] = 0) & (OwnershipState[14] = 0) &
			(OwnershipState[15] = 0) & (OwnershipState[16] = 0) &
			(OwnershipState[17] = 0) & (OwnershipState[18] = 0) &
			(OwnershipState[19] = 0) & (OwnershipState[20] = 0) &
			(OwnershipState[21] = 0) & (OwnershipState[24] = 0) &
			(OwnershipState[25] = 0) & (OwnershipState[26] = 0) &
			(OwnershipState[27] = 0);
		axisIndex := 1;
		while axisIndex <= LMC_OWNER_AXIS_COUNT do
			recordBase := LMC_OWNER_GLOBAL_SLOTS +
				((axisIndex - 1) * LMC_OWNER_AXIS_STRIDE);
			if (OwnershipState[recordBase] <> axisIndex) |
				(OwnershipState[recordBase + 35]$UDINT <>
				 (LMC_OWNER_AXIS_RECORD_MAGIC + TO_UDINT(axisIndex))) then
				tableIdle := FALSE;
			end_if;
			stateIndex := 1;
			while stateIndex <= 34 do
				if OwnershipState[recordBase + stateIndex] <> 0 then
					tableIdle := FALSE;
				end_if;
				stateIndex += 1;
			end_while;
			axisIndex += 1;
		end_while;
		if tableIdle = FALSE then
			Result := -3;
			RETURN;
		end_if;
	else
		Result := -3;
		RETURN;
	end_if;

	if (OwnershipStartupState[0]$UDINT <> LMC_OWNER_STARTUP_STATE_MAGIC) |
		(OwnershipStartupState[1]$UDINT <> DiagnosticsBootId) then
		_memset(dest:=#OwnershipStartupState[0], usByte:=0, cntr:=64);
		OwnershipStartupState[0]$UDINT := LMC_OWNER_STARTUP_STATE_MAGIC;
		OwnershipStartupState[1]$UDINT := DiagnosticsBootId;
	end_if;

	Result := 1;
	if IsClientConnected(#InputLatch) = FALSE then
		OwnershipStartupState[3] := 0;
		OwnershipStartupState[4]$UDINT := 0x00000001;
		OwnershipStartupState[14] := 0;
		OwnershipStartupState[15] := 1;
		RETURN;
	end_if;
	copyResult := InputLatch.CopyAxisOwnershipStartupSnapshot(
		pDest:=#startupSnapshot[0], DestSize:=48);
	if copyResult <> 0 then
		OwnershipStartupState[3] := 0;
		OwnershipStartupState[4]$UDINT := 0x00000001;
		OwnershipStartupState[14] := 0;
		OwnershipStartupState[15] := 2;
		RETURN;
	end_if;
	if (startupSnapshot[0] <> LMC_OWNER_STARTUP_SNAPSHOT_MAGIC) |
		(startupSnapshot[1] = 0) |
		(startupSnapshot[1] <> ObservationCycle) |
		(startupSnapshot[11] <> 0) then
		OwnershipStartupState[3] := 0;
		OwnershipStartupState[14] := 0;
		OwnershipStartupState[15] := -1;
		Result := -1;
		RETURN;
	end_if;

	physicalIdle :=
		((startupSnapshot[10] and 0x00000001) <> 0) &
		((startupSnapshot[2] and LMC_AXIS_STATUS_STANDSTILL) <> 0) &
		((startupSnapshot[2] and LMC_OWNER_STARTUP_AXIS_CLEAR_MASK) = 0) &
		((startupSnapshot[3] and LMC_AXIS_STATUS_STANDSTILL) <> 0) &
		((startupSnapshot[3] and LMC_OWNER_STARTUP_AXIS_CLEAR_MASK) = 0) &
		((startupSnapshot[4] and LMC_AXIS_STATUS_STANDSTILL) <> 0) &
		((startupSnapshot[4] and LMC_OWNER_STARTUP_AXIS_CLEAR_MASK) = 0) &
		((startupSnapshot[5] and LMC_AXIS_STATUS_STANDSTILL) <> 0) &
		((startupSnapshot[5] and LMC_OWNER_STARTUP_AXIS_CLEAR_MASK) = 0);

	groupIdle := FALSE;
	groupSignature := 0;
	if (IsClientConnected(#LMCRobot) <> 0) &
		(IsClientConnected(#LMCAxis1) <> 0) &
		(IsClientConnected(#LMCAxis2) <> 0) &
		(IsClientConnected(#LMCAxis3) <> 0) &
		(IsClientConnected(#LMCAxis4) <> 0) then
		robotState := LMCRobot.ReadRobotParameter(ParNo:=_ROBOT_STATE, Mode:=0);
		profileLockState := LMCRobot.ReadProfileParameter(
			ParNo:=_LMCPROF_LockState);
		profileFinished := LMCRobot.ProfileInPosition(
			Mode:=_LMCPROF_ProfileFinished);
		groupSignature := (TO_UDINT(robotState) and 0x0000FFFF) or
			((TO_UDINT(profileLockState) and 0x000000FF) shl 16);
		if profileFinished <> 0 then
			groupSignature := groupSignature or 0x01000000;
		end_if;
		groupIdle := (profileLockState = 0) &
			((startupSnapshot[2] and LMC_OWNER_STARTUP_AXIS_LOCK_MASK) = 0) &
			((startupSnapshot[3] and LMC_OWNER_STARTUP_AXIS_LOCK_MASK) = 0) &
			((startupSnapshot[4] and LMC_OWNER_STARTUP_AXIS_LOCK_MASK) = 0) &
			((startupSnapshot[5] and LMC_OWNER_STARTUP_AXIS_LOCK_MASK) = 0) &
			((robotState = _ROBOT_PASSIVE$DINT) |
			 ((robotState = _ROBOT_DIRECT$DINT) & (profileFinished <> 0)));
	end_if;

	drained := (startupSnapshot[10] = LMC_OWNER_STARTUP_LATCH_REQUIRED) &
		(DiagnosticsDrainFlags = LMC_OWNER_STARTUP_DIAG_REQUIRED) &
		(ZeroHomeState[0] <> LMC_HOME_RECORD_RUNNING) &
		(ZeroHomeState[0] <> LMC_HOME_RECORD_QUARANTINED) &
		((ZeroHomeState[39] = LMC_HOME_ENGINE_IDLE) |
		 (ZeroHomeState[39] = LMC_HOME_ENGINE_TERMINAL));

	combinedProof := 0x00000001;
	if physicalIdle then
		combinedProof := combinedProof or 0x00000002;
	end_if;
	if groupIdle then
		combinedProof := combinedProof or 0x00000004;
	end_if;
	if drained then
		combinedProof := combinedProof or 0x00000008;
	end_if;

	if combinedProof <> LMC_OWNER_STARTUP_PROOF_REQUIRED then
		OwnershipStartupState[2]$UDINT := ObservationCycle;
		OwnershipStartupState[3] := 0;
		OwnershipStartupState[4]$UDINT := combinedProof;
		OwnershipStartupState[5]$UDINT := groupSignature;
		OwnershipStartupState[6]$UDINT := startupSnapshot[2];
		OwnershipStartupState[7]$UDINT := startupSnapshot[3];
		OwnershipStartupState[8]$UDINT := startupSnapshot[4];
		OwnershipStartupState[9]$UDINT := startupSnapshot[5];
		OwnershipStartupState[10]$UDINT := startupSnapshot[6];
		OwnershipStartupState[11]$UDINT := startupSnapshot[7];
		OwnershipStartupState[12]$UDINT := startupSnapshot[8];
		OwnershipStartupState[13]$UDINT := startupSnapshot[9];
		OwnershipStartupState[14] := 0;
		OwnershipStartupState[15] := 3;
		RETURN;
	end_if;

	signatureStable :=
		(OwnershipStartupState[4]$UDINT = combinedProof) &
		(OwnershipStartupState[5]$UDINT = groupSignature) &
		(OwnershipStartupState[6]$UDINT = startupSnapshot[2]) &
		(OwnershipStartupState[7]$UDINT = startupSnapshot[3]) &
		(OwnershipStartupState[8]$UDINT = startupSnapshot[4]) &
		(OwnershipStartupState[9]$UDINT = startupSnapshot[5]) &
		(OwnershipStartupState[10]$UDINT = startupSnapshot[6]) &
		(OwnershipStartupState[11]$UDINT = startupSnapshot[7]) &
		(OwnershipStartupState[12]$UDINT = startupSnapshot[8]) &
		(OwnershipStartupState[13]$UDINT = startupSnapshot[9]);

	freshObservation := FALSE;
	if OwnershipStartupState[3] <= 0 then
		OwnershipStartupState[3] := 1;
		OwnershipStartupState[14]$UDINT := ReportCycle;
		freshObservation := TRUE;
	elsif OwnershipStartupState[2]$UDINT <> ObservationCycle then
		freshObservation := TRUE;
		if signatureStable then
			if OwnershipStartupState[3] < LMC_OWNER_STARTUP_STABLE_SAMPLES then
				OwnershipStartupState[3] += 1;
			end_if;
		else
			OwnershipStartupState[3] := 1;
			OwnershipStartupState[14]$UDINT := ReportCycle;
		end_if;
	elsif signatureStable = FALSE then
		OwnershipStartupState[3] := 0;
		OwnershipStartupState[14] := 0;
		OwnershipStartupState[15] := 4;
	end_if;

	OwnershipStartupState[2]$UDINT := ObservationCycle;
	OwnershipStartupState[4]$UDINT := combinedProof;
	OwnershipStartupState[5]$UDINT := groupSignature;
	OwnershipStartupState[6]$UDINT := startupSnapshot[2];
	OwnershipStartupState[7]$UDINT := startupSnapshot[3];
	OwnershipStartupState[8]$UDINT := startupSnapshot[4];
	OwnershipStartupState[9]$UDINT := startupSnapshot[5];
	OwnershipStartupState[10]$UDINT := startupSnapshot[6];
	OwnershipStartupState[11]$UDINT := startupSnapshot[7];
	OwnershipStartupState[12]$UDINT := startupSnapshot[8];
	OwnershipStartupState[13]$UDINT := startupSnapshot[9];
	if OwnershipStartupState[3] > 0 then
		OwnershipStartupState[15] := 0;
	end_if;

	if OwnershipStartupState[3] < LMC_OWNER_STARTUP_STABLE_SAMPLES then
		RETURN;
	end_if;
	if freshObservation = FALSE then
		RETURN;
	end_if;
	stableElapsedMilliseconds := ReportCycle -
		OwnershipStartupState[14]$UDINT;
	if stableElapsedMilliseconds < LMC_OWNER_STARTUP_STABLE_MS then
		RETURN;
	end_if;

	_memset(dest:=#OwnershipState[0], usByte:=0, cntr:=1408);
	_memset(dest:=#OwnershipObserverState[0], usByte:=0, cntr:=432);
	_memset(dest:=#OwnershipLeaseState[0], usByte:=0,
		cntr:=sizeof(OwnershipLeaseState));
	_memset(dest:=#OwnershipPreemptedState[0], usByte:=0,
		cntr:=sizeof(OwnershipPreemptedState));
	_memset(dest:=#OwnershipIdentityState[0], usByte:=0,
		cntr:=sizeof(OwnershipIdentityState));
	_memset(dest:=#OwnershipLeaseIdentityState[0], usByte:=0,
		cntr:=sizeof(OwnershipLeaseIdentityState));
	_memset(dest:=#OwnershipPreemptedIdentityState[0], usByte:=0,
		cntr:=sizeof(OwnershipPreemptedIdentityState));
	OwnershipState[0]$UDINT := LMC_OWNER_TABLE_MAGIC;
	OwnershipState[3]$UDINT := DiagnosticsBootId;
	OwnershipState[4]$UDINT := ReportCycle;
	OwnershipState[5]$UDINT := LMC_OWNER_STARTUP_PROOF_REQUIRED;
	axisIndex := 1;
	while axisIndex <= LMC_OWNER_AXIS_COUNT do
		recordBase := LMC_OWNER_GLOBAL_SLOTS +
			((axisIndex - 1) * LMC_OWNER_AXIS_STRIDE);
		OwnershipState[recordBase] := axisIndex;
		OwnershipState[recordBase + 35]$UDINT :=
			LMC_OWNER_AXIS_RECORD_MAGIC + TO_UDINT(axisIndex);
		axisIndex += 1;
	end_while;
	Result := 0;

END_FUNCTION

FUNCTION GLOBAL LMCControlCommandService::NotifyAxisOwnershipSessionClosed
	VAR_INPUT
		SessionEpoch : UDINT;
	END_VAR
	VAR
		axisIndex : DINT;
		axisBit : UDINT;
		recordBase : DINT;
	END_VAR

	if SessionEpoch = 0 then
		RETURN;
	end_if;
	if (SessionEpoch <> 0) &
	   (AxisSetPositionAsyncState[3]$UDINT = SessionEpoch) &
	   ((AxisSetPositionAsyncState[1] =
	     LMC_ADMIN_SET_POSITION_ASYNC_STATE_OWNERSHIP_RESERVED) |
	    (AxisSetPositionAsyncState[1] =
	     LMC_ADMIN_SET_POSITION_ASYNC_STATE_PREFLIGHT_PENDING) |
	    (AxisSetPositionAsyncState[1] =
	     LMC_ADMIN_SET_POSITION_ASYNC_STATE_PREFLIGHT_READY) |
	    (AxisSetPositionAsyncState[1] =
	     LMC_ADMIN_SET_POSITION_ASYNC_STATE_OWNERSHIP_ACTIVE)) then
		AxisSetPositionAsyncState[1] :=
			LMC_ADMIN_SET_POSITION_ASYNC_STATE_QUARANTINED;
		AxisSetPositionAsyncState[31] := 2;
	end_if;
	OwnershipState[22]$UDINT := SessionEpoch;
	axisIndex := 1;
	while axisIndex <= LMC_OWNER_AXIS_COUNT do
		case axisIndex of
			1: axisBit := 0x00000001;
			2: axisBit := 0x00000002;
			3: axisBit := 0x00000004;
			4: axisBit := 0x00000008;
			5: axisBit := 0x00000010;
			6: axisBit := 0x00000020;
			7: axisBit := 0x00000040;
			8: axisBit := 0x00000080;
			9: axisBit := 0x00000100;
		else
			axisBit := 0;
		end_case;
		recordBase := LMC_OWNER_GLOBAL_SLOTS +
			((axisIndex - 1) * LMC_OWNER_AXIS_STRIDE);
		if (OwnershipState[recordBase + 6]$UDINT = SessionEpoch) &
		   ((OwnershipState[recordBase + 1] = LMC_OWNER_STATE_RESERVED) |
		    ((OwnershipState[recordBase + 1] =
		      LMC_OWNER_STATE_DIRECT_ACTIVE) &
		     (AxisSetPositionAsyncState[0]$UDINT =
		      LMC_ADMIN_SET_POSITION_ASYNC_MAGIC) &
		     (AxisSetPositionAsyncState[1] =
		      LMC_ADMIN_SET_POSITION_ASYNC_STATE_QUARANTINED) &
		     (OwnershipState[recordBase + 2] = LMC_OWNER_KIND_DIRECT) &
		     (OwnershipState[recordBase + 3] = 0x7D12) &
		     (OwnershipState[recordBase + 4]$UDINT =
		      AxisSetPositionAsyncState[5]$UDINT) &
		     (OwnershipState[recordBase + 5]$UDINT =
		      AxisSetPositionAsyncState[6]$UDINT) &
		     (OwnershipState[recordBase + 7]$UDINT =
		      AxisSetPositionAsyncState[4]$UDINT) &
		     (OwnershipState[recordBase + 11]$UDINT = axisBit) &
		     (OwnershipState[recordBase + 11]$UDINT =
		      AxisSetPositionAsyncState[7]$UDINT) &
		     (OwnershipState[recordBase + 12] =
		      AxisSetPositionAsyncState[11]))) then
			OwnershipState[recordBase + 1] := LMC_OWNER_STATE_QUARANTINED;
			OwnershipState[recordBase + 32] :=
				LMC_OWNER_REPORT_QUARANTINE;
			OwnershipState[recordBase + 33] := -20;
		end_if;
		axisIndex += 1;
	end_while;

END_FUNCTION

FUNCTION GLOBAL LMCControlCommandService::ProcessAxisOwnership
	VAR
		latchSnapshot : ARRAY [0..303] OF USINT;
		startupSnapshot : ARRAY [0..11] OF UDINT;
		axisIndex : DINT;
		selectedAxisIndex : DINT;
		leaderAxisIndex : DINT;
		axisBit : UDINT;
		selectedAxisBit : UDINT;
		recordBase : DINT;
		selectedRecordBase : DINT;
		observerBase : DINT;
		selectedObserverBase : DINT;
		axisMask : UDINT;
		admissionToken : UDINT;
		ownerGeneration : UDINT;
		latchCycle : UDINT;
		serviceNow : UDINT;
		stableElapsed : UDINT;
		ownerElapsed : UDINT;
		commandId : DINT;
		ownerReference : DINT;
		ownerKind : DINT;
		ownerState : DINT;
		admissionMode : DINT;
		axisStatusRaw : UDINT;
		axisErrorRaw : UDINT;
		ds402StatusRaw : UDINT;
		profileErrorInfo : _LMCPROFERRORDEF;
		groupPowerState : DINT;
		groupLockState : DINT;
		groupFinished : DINT;
		groupError : DINT;
		latchCopyResult : DINT;
		startupCopyResult : DINT;
		publishResult : DINT;
		reportKind : UINT;
		allConnected : BOOL;
		allStandstill : BOOL;
		allPowerOn : BOOL;
		allPowerOff : BOOL;
		allErrorClear : BOOL;
		allTargetReached : BOOL;
		referencePowerOff : BOOL;
		powerOffEscalated : BOOL;
		tupleValid : BOOL;
		coherentObservation : BOOL;
		freshObservation : BOOL;
		terminalCandidate : BOOL;
		safeFailure : BOOL;
		forceQuarantine : BOOL;
		activitySeen : BOOL;
		unsupportedAxisSelected : BOOL;
	END_VAR

	if OwnershipState[0]$UDINT <> LMC_OWNER_TABLE_MAGIC then
		RETURN;
	end_if;
	OwnershipState[23]$UDINT := ops.tAbsolute;
	axisIndex := 1;
	while axisIndex <= LMC_OWNER_AXIS_COUNT do
		recordBase := LMC_OWNER_GLOBAL_SLOTS +
			((axisIndex - 1) * LMC_OWNER_AXIS_STRIDE);
		if OwnershipState[recordBase + 35]$UDINT <>
		   (LMC_OWNER_AXIS_RECORD_MAGIC + TO_UDINT(axisIndex)) then
			OwnershipState[24] := 1;
			OwnershipState[recordBase + 1] :=
				LMC_OWNER_STATE_QUARANTINED;
		end_if;
		axisIndex += 1;
	end_while;
	if LMC_AXIS_OWNERSHIP_ORDINARY_ENABLED = FALSE then
		RETURN;
	end_if;

	latchCopyResult := -1;
	startupCopyResult := -1;
	coherentObservation := FALSE;
	latchCycle := 0;
	if IsClientConnected(#InputLatch) then
		latchCopyResult := InputLatch.CopySnapshot(
			pDest:=#latchSnapshot[0], DestSize:=304);
		startupCopyResult := InputLatch.CopyAxisOwnershipStartupSnapshot(
			pDest:=#startupSnapshot[0], DestSize:=48);
	end_if;
	if (latchCopyResult = 0) & (startupCopyResult = 0) then
		latchCycle := latchSnapshot[0]$UDINT;
		coherentObservation :=
			(startupSnapshot[0] = LMC_OWNER_STARTUP_SNAPSHOT_MAGIC) &
			(latchCycle <> 0) & (startupSnapshot[1] = latchCycle) &
			((startupSnapshot[10] and
			  LMC_OWNER_LATCH_PHYSICAL_FLAG) <> 0) &
			(startupSnapshot[11] = 0) &
			(latchSnapshot[84]$UDINT = startupSnapshot[6]) &
			(latchSnapshot[120]$UDINT = startupSnapshot[7]) &
			(latchSnapshot[156]$UDINT = startupSnapshot[8]) &
			(latchSnapshot[192]$UDINT = startupSnapshot[9]);
	end_if;
	if coherentObservation = FALSE then
		latchCycle := 0;
	end_if;

	serviceNow := ops.tAbsolute;
	if serviceNow = 0 then
		serviceNow := 1;
	end_if;
	axisIndex := 1;
	while axisIndex <= LMC_OWNER_AXIS_COUNT do
		case axisIndex of
			1: axisBit := 0x00000001;
			2: axisBit := 0x00000002;
			3: axisBit := 0x00000004;
			4: axisBit := 0x00000008;
			5: axisBit := 0x00000010;
			6: axisBit := 0x00000020;
			7: axisBit := 0x00000040;
			8: axisBit := 0x00000080;
			9: axisBit := 0x00000100;
		else
			axisBit := 0;
		end_case;
		recordBase := LMC_OWNER_GLOBAL_SLOTS +
			((axisIndex - 1) * LMC_OWNER_AXIS_STRIDE);
		ownerState := OwnershipState[recordBase + 1];
		ownerKind := OwnershipState[recordBase + 2];
		if ((ownerKind = LMC_OWNER_KIND_DIRECT) |
		    (ownerKind = LMC_OWNER_KIND_GROUP)) &
		   ((ownerState = LMC_OWNER_STATE_DIRECT_ACTIVE) |
		    (ownerState = LMC_OWNER_STATE_GROUP_ACTIVE) |
		    (ownerState = LMC_OWNER_STATE_SAFETY_PREEMPTING)) &
		   (OwnershipState[recordBase + 3] <> 0x7D12) then
			axisMask := OwnershipState[recordBase + 11]$UDINT;
			admissionToken := OwnershipState[recordBase + 4]$UDINT;
			ownerGeneration := OwnershipState[recordBase + 5]$UDINT;
			commandId := OwnershipState[recordBase + 3];
			ownerReference := OwnershipState[recordBase + 12];
			admissionMode := OwnershipState[recordBase + 14];
			leaderAxisIndex := 0;
			if (axisMask and 0x00000001) <> 0 then
				leaderAxisIndex := 1;
			elsif (axisMask and 0x00000002) <> 0 then
				leaderAxisIndex := 2;
			elsif (axisMask and 0x00000004) <> 0 then
				leaderAxisIndex := 3;
			elsif (axisMask and 0x00000008) <> 0 then
				leaderAxisIndex := 4;
			elsif (axisMask and 0x00000010) <> 0 then
				leaderAxisIndex := 5;
			elsif (axisMask and 0x00000020) <> 0 then
				leaderAxisIndex := 6;
			elsif (axisMask and 0x00000040) <> 0 then
				leaderAxisIndex := 7;
			elsif (axisMask and 0x00000080) <> 0 then
				leaderAxisIndex := 8;
			elsif (axisMask and 0x00000100) <> 0 then
				leaderAxisIndex := 9;
			end_if;

			if axisIndex = leaderAxisIndex then
				observerBase := (axisIndex - 1) * LMC_OWNER_OBSERVER_STRIDE;
				powerOffEscalated :=
					(OwnershipObserverState[observerBase + 5]$UDINT and
					 LMC_OWNER_OBSERVER_POWER_OFF_ESCALATED) <> 0;
				tupleValid := (axisMask <> 0) &
					(axisMask <= LMC_OWNER_ROBOT_AXIS_MASK) &
					(admissionToken <> 0) & (ownerGeneration <> 0);
				forceQuarantine := FALSE;
				unsupportedAxisSelected :=
					(axisMask and LMC_OWNER_UNSUPPORTED_AXIS_MASK) <> 0;
				selectedAxisIndex := 1;
				while selectedAxisIndex <= LMC_OWNER_AXIS_COUNT do
					case selectedAxisIndex of
						1: selectedAxisBit := 0x00000001;
						2: selectedAxisBit := 0x00000002;
						3: selectedAxisBit := 0x00000004;
						4: selectedAxisBit := 0x00000008;
						5: selectedAxisBit := 0x00000010;
						6: selectedAxisBit := 0x00000020;
						7: selectedAxisBit := 0x00000040;
						8: selectedAxisBit := 0x00000080;
						9: selectedAxisBit := 0x00000100;
					else
						selectedAxisBit := 0;
					end_case;
					selectedRecordBase := LMC_OWNER_GLOBAL_SLOTS +
						((selectedAxisIndex - 1) * LMC_OWNER_AXIS_STRIDE);
					selectedObserverBase :=
						(selectedAxisIndex - 1) * LMC_OWNER_OBSERVER_STRIDE;
					if (axisMask and selectedAxisBit) <> 0 then
						if (OwnershipState[selectedRecordBase + 1] <>
						    ownerState) |
						   (OwnershipState[selectedRecordBase + 2] <> ownerKind) |
						   (OwnershipState[selectedRecordBase + 3] <> commandId) |
						   (OwnershipState[selectedRecordBase + 4]$UDINT <>
						    admissionToken) |
						   (OwnershipState[selectedRecordBase + 5]$UDINT <>
						    ownerGeneration) |
						   (OwnershipState[selectedRecordBase + 11]$UDINT <>
						    axisMask) |
						   (OwnershipObserverState[selectedObserverBase]$UDINT <>
						    (LMC_OWNER_OBSERVER_MAGIC +
						     TO_UDINT(selectedAxisIndex))) |
						   (OwnershipObserverState[selectedObserverBase + 1]$UDINT <>
						    admissionToken) |
						   (OwnershipObserverState[selectedObserverBase + 2]$UDINT <>
						    ownerGeneration) |
						   (((OwnershipObserverState[selectedObserverBase + 5]$UDINT and
						      LMC_OWNER_OBSERVER_POWER_OFF_ESCALATED) <> 0) <>
						    powerOffEscalated) then
							tupleValid := FALSE;
						end_if;
						if (OwnershipObserverState[selectedObserverBase + 5]$UDINT and
						    LMC_OWNER_OBSERVER_FORCE_QUARANTINE) <> 0 then
							forceQuarantine := TRUE;
						end_if;
					end_if;
					selectedAxisIndex += 1;
				end_while;
				if powerOffEscalated &
				   (commandId <> LMC_OWNER_COMMAND_AXIS_STOP) &
				   (commandId <> LMC_OWNER_COMMAND_GROUP_DISABLE) &
				   (commandId <> LMC_OWNER_COMMAND_GROUP_STOP) then
					tupleValid := FALSE;
				end_if;

				if tupleValid = FALSE then
					OwnershipState[24] := 1;
					selectedAxisIndex := 1;
					while selectedAxisIndex <= LMC_OWNER_AXIS_COUNT do
						case selectedAxisIndex of
							1: selectedAxisBit := 0x00000001;
							2: selectedAxisBit := 0x00000002;
							3: selectedAxisBit := 0x00000004;
							4: selectedAxisBit := 0x00000008;
							5: selectedAxisBit := 0x00000010;
							6: selectedAxisBit := 0x00000020;
							7: selectedAxisBit := 0x00000040;
							8: selectedAxisBit := 0x00000080;
							9: selectedAxisBit := 0x00000100;
						else
							selectedAxisBit := 0;
						end_case;
						if (axisMask and selectedAxisBit) <> 0 then
							selectedRecordBase := LMC_OWNER_GLOBAL_SLOTS +
								((selectedAxisIndex - 1) *
								 LMC_OWNER_AXIS_STRIDE);
							OwnershipState[selectedRecordBase + 1] :=
								LMC_OWNER_STATE_QUARANTINED;
							OwnershipState[selectedRecordBase + 32] :=
								LMC_OWNER_REPORT_QUARANTINE;
							OwnershipState[selectedRecordBase + 33] := -24;
						end_if;
						selectedAxisIndex += 1;
					end_while;
				elsif unsupportedAxisSelected then
					publishResult := PublishAxisOwnership(
						AxisMask:=axisMask,
						AdmissionToken:=admissionToken,
						OwnerGeneration:=ownerGeneration,
						ReportKind:=LMC_OWNER_REPORT_QUARANTINE,
						ReportValue0:=TO_UDINT(commandId),
						ReportValue1:=axisMask and
							LMC_OWNER_UNSUPPORTED_AXIS_MASK,
						ObservationCycle:=0);
					if publishResult <> 0 then
						OwnershipState[24] := 1;
					end_if;
				else
					observerBase := (axisIndex - 1) * LMC_OWNER_OBSERVER_STRIDE;
					freshObservation := coherentObservation &
						OwnershipObserverState[observerBase + 8]$UDINT <>
						latchCycle;
					reportKind := 0;
					groupError := 0;
					ownerElapsed := serviceNow -
						OwnershipState[recordBase + 8]$UDINT;
					if coherentObservation = FALSE then
						OwnershipObserverState[observerBase + 3] := 0;
						OwnershipObserverState[observerBase + 4] := 0;
						OwnershipObserverState[observerBase + 5]$UDINT :=
							OwnershipObserverState[observerBase + 5]$UDINT and
							LMC_OWNER_OBSERVER_EVIDENCE_CLEAR_MASK;
						OwnershipObserverState[observerBase + 6] := 0;
						OwnershipObserverState[observerBase + 7] := 0;
					end_if;
					if freshObservation then
						allConnected := TRUE;
						allStandstill := TRUE;
						allPowerOn := TRUE;
						allPowerOff := TRUE;
						allErrorClear := TRUE;
						allTargetReached := TRUE;
						referencePowerOff := FALSE;
						activitySeen :=
							(OwnershipObserverState[observerBase + 5]$UDINT and
							 LMC_OWNER_OBSERVER_ACTIVITY_SEEN) <> 0;
						selectedAxisIndex := 1;
						while selectedAxisIndex <= LMC_OWNER_AXIS_COUNT do
							case selectedAxisIndex of
								1: selectedAxisBit := 0x00000001;
								2: selectedAxisBit := 0x00000002;
								3: selectedAxisBit := 0x00000004;
								4: selectedAxisBit := 0x00000008;
								5: selectedAxisBit := 0x00000010;
								6: selectedAxisBit := 0x00000020;
								7: selectedAxisBit := 0x00000040;
								8: selectedAxisBit := 0x00000080;
								9: selectedAxisBit := 0x00000100;
							else
								selectedAxisBit := 0;
							end_case;
							if (axisMask and selectedAxisBit) <> 0 then
								axisStatusRaw := 0;
								axisErrorRaw := 0;
								ds402StatusRaw := 0;
								case selectedAxisIndex of
									1:
										axisStatusRaw := startupSnapshot[2];
										ds402StatusRaw := startupSnapshot[6];
										axisErrorRaw := TO_UDINT(
											latchSnapshot[88]$DINT);
									2:
										axisStatusRaw := startupSnapshot[3];
										ds402StatusRaw := startupSnapshot[7];
										axisErrorRaw := TO_UDINT(
											latchSnapshot[124]$DINT);
									3:
										axisStatusRaw := startupSnapshot[4];
										ds402StatusRaw := startupSnapshot[8];
										axisErrorRaw := TO_UDINT(
											latchSnapshot[160]$DINT);
									4:
										axisStatusRaw := startupSnapshot[5];
										ds402StatusRaw := startupSnapshot[9];
										axisErrorRaw := TO_UDINT(
											latchSnapshot[196]$DINT);
								else
									allConnected := FALSE;
								end_case;
								if (axisStatusRaw and
								    LMC_AXIS_STATUS_STANDSTILL) = 0 then
									allStandstill := FALSE;
									activitySeen := TRUE;
								end_if;
								if ((axisStatusRaw and
								     LMC_OWNER_AXIS_POWER_ON_MASK) = 0) |
								   ((ds402StatusRaw and LMC_OWNER_DS402_STATE_MASK) <>
								    LMC_OWNER_DS402_OPERATION_ENABLED_STATE) then
									allPowerOn := FALSE;
								end_if;
								if ((axisStatusRaw and
								     LMC_OWNER_AXIS_POWER_ON_MASK) <> 0) |
								   ((ds402StatusRaw and
								     LMC_OWNER_DS402_OPERATION_ENABLED_MASK) <> 0) then
									allPowerOff := FALSE;
								end_if;
								if selectedAxisIndex = ownerReference then
									referencePowerOff :=
										((axisStatusRaw and
										  LMC_OWNER_AXIS_POWER_ON_MASK) = 0) &
										((ds402StatusRaw and
										  LMC_OWNER_DS402_OPERATION_ENABLED_MASK) = 0);
								end_if;
								if (axisErrorRaw <> 0) |
								   ((axisStatusRaw and
								     LMC_OWNER_AXIS_EMERGENCY_MASK) <> 0) |
								   ((ds402StatusRaw and
								     LMC_OWNER_DS402_FAULT_MASK) <> 0) then
									allErrorClear := FALSE;
								end_if;
								if (ds402StatusRaw and
								    LMC_OWNER_DS402_TARGET_REACHED_MASK) = 0 then
									allTargetReached := FALSE;
								end_if;
								if selectedAxisIndex = leaderAxisIndex then
									if (OwnershipObserverState[observerBase + 5]$UDINT and
									    LMC_OWNER_OBSERVER_BASELINE_VALID) = 0 then
										OwnershipObserverState[observerBase + 3]$UDINT :=
											axisStatusRaw;
										OwnershipObserverState[observerBase + 4]$UDINT :=
											ds402StatusRaw;
										OwnershipObserverState[observerBase + 5]$UDINT :=
											OwnershipObserverState[observerBase + 5]$UDINT or
											LMC_OWNER_OBSERVER_BASELINE_VALID;
									elsif ((axisStatusRaw and
									        LMC_OWNER_AXIS_IN_POSITION_MASK) <>
									       (OwnershipObserverState[observerBase + 3]$UDINT and
									        LMC_OWNER_AXIS_IN_POSITION_MASK)) |
									      ((ds402StatusRaw and
									        LMC_OWNER_DS402_TARGET_REACHED_MASK) <>
									       (OwnershipObserverState[observerBase + 4]$UDINT and
									        LMC_OWNER_DS402_TARGET_REACHED_MASK)) then
										activitySeen := TRUE;
									end_if;
								end_if;
							end_if;
							selectedAxisIndex += 1;
						end_while;

						groupPowerState := 0;
						groupLockState := 0;
						groupFinished := 0;
						groupError := 0;
						if ownerKind = LMC_OWNER_KIND_GROUP then
							if IsClientConnected(#LMCRobot) then
								groupPowerState := LMCRobot.RobotIsOn();
								groupLockState := LMCRobot.ReadProfileParameter(
									ParNo:=_LMCPROF_LockState);
								groupFinished := LMCRobot.ProfileInPosition(
									Mode:=_LMCPROF_ProfileFinished);
								profileErrorInfo := LMCRobot.ReadProfileError();
								groupError := TO_DINT(profileErrorInfo.ErrorNo);
							else
								allConnected := FALSE;
							end_if;
							if groupFinished = 0 then
								activitySeen := TRUE;
							end_if;
						end_if;

						if activitySeen then
							OwnershipObserverState[observerBase + 5]$UDINT :=
								OwnershipObserverState[observerBase + 5]$UDINT or
								LMC_OWNER_OBSERVER_ACTIVITY_SEEN;
						end_if;
						terminalCandidate := FALSE;
						safeFailure := FALSE;
						if allConnected then
							if ownerKind = LMC_OWNER_KIND_DIRECT then
								case commandId of
									0x2023:
										if admissionMode =
										   LMC_OWNER_ADMISSION_SAFETY then
											terminalCandidate := allPowerOff;
										else
											terminalCandidate := allPowerOn &
												allErrorClear;
										end_if;
									0x2024:
										terminalCandidate := allErrorClear;
									0x2022:
										if powerOffEscalated then
											terminalCandidate := referencePowerOff;
										else
											terminalCandidate := allStandstill;
										end_if;
									0x209F, 0x20A0:
										terminalCandidate := activitySeen & allStandstill &
											allTargetReached;
									0x20A2:
										terminalCandidate := FALSE;
								else
									forceQuarantine := TRUE;
								end_case;
							else
								case commandId of
									0x2047:
										terminalCandidate :=
											(groupLockState <> 0) &
											(groupFinished <> 0) & allStandstill &
											allPowerOn & allErrorClear &
											(groupError = 0);
									0x2048:
										if powerOffEscalated then
											terminalCandidate :=
												(groupPowerState = 0) & allPowerOff;
										else
											terminalCandidate :=
												(groupLockState = 0) &
												(groupFinished <> 0) & allStandstill;
										end_if;
									0x2049:
										terminalCandidate :=
											allErrorClear & (groupError = 0);
									0x204A:
										terminalCandidate :=
											(groupPowerState <> 0) & allPowerOn &
											allErrorClear & (groupError = 0);
									0x204B:
										terminalCandidate :=
											(groupPowerState = 0) & allPowerOff;
									0x2085:
										if powerOffEscalated then
											terminalCandidate :=
												(groupPowerState = 0) & allPowerOff;
										else
											terminalCandidate :=
												(groupFinished <> 0) & allStandstill;
										end_if;
									0x20A4, 0x7D22:
										terminalCandidate := activitySeen &
											(groupFinished <> 0) & allStandstill &
											allTargetReached;
								else
									forceQuarantine := TRUE;
								end_case;
							end_if;
						end_if;
						if terminalCandidate &
						   ((allErrorClear = FALSE) | (groupError <> 0)) then
							safeFailure := TRUE;
						end_if;

						if terminalCandidate then
							if OwnershipObserverState[observerBase + 6] <= 0 then
								OwnershipObserverState[observerBase + 6] := 1;
								OwnershipObserverState[observerBase + 7]$UDINT :=
									serviceNow;
							elsif OwnershipObserverState[observerBase + 6] <
							      LMC_OWNER_ORDINARY_STABLE_SAMPLES then
								OwnershipObserverState[observerBase + 6] += 1;
							end_if;
						else
							OwnershipObserverState[observerBase + 6] := 0;
							OwnershipObserverState[observerBase + 7] := 0;
						end_if;
						OwnershipObserverState[observerBase + 8]$UDINT := latchCycle;
						OwnershipState[recordBase + 9]$UDINT := latchCycle;
						OwnershipState[recordBase + 10]$UDINT :=
							OwnershipObserverState[observerBase + 7]$UDINT;

						stableElapsed := 0;
						if OwnershipObserverState[observerBase + 7]$UDINT <> 0 then
							stableElapsed := serviceNow -
								OwnershipObserverState[observerBase + 7]$UDINT;
						end_if;
						if terminalCandidate &
						   (OwnershipObserverState[observerBase + 6] >=
						    LMC_OWNER_ORDINARY_STABLE_SAMPLES) &
						   (stableElapsed >= LMC_OWNER_ORDINARY_STABLE_MS) then
							if forceQuarantine then
								reportKind := LMC_OWNER_REPORT_QUARANTINE;
							elsif safeFailure then
								reportKind :=
									LMC_OWNER_REPORT_TERMINAL_SAFE_FAILURE;
							else
								reportKind := LMC_OWNER_REPORT_TERMINAL_SUCCESS;
							end_if;
						end_if;
					end_if;
					if (reportKind = 0) & (commandId <> 0x20A2) &
					   (ownerElapsed > LMC_OWNER_ORDINARY_TIMEOUT_MS) then
						reportKind := LMC_OWNER_REPORT_QUARANTINE;
					end_if;
					if reportKind <> 0 then
						publishResult := PublishAxisOwnership(
							AxisMask:=axisMask,
							AdmissionToken:=admissionToken,
							OwnerGeneration:=ownerGeneration,
							ReportKind:=reportKind,
							ReportValue0:=TO_UDINT(commandId),
							ReportValue1:=TO_UDINT(groupError),
							ObservationCycle:=latchCycle);
						if publishResult <> 0 then
							OwnershipState[24] := 1;
						end_if;
					end_if;
				end_if;
			end_if;
		end_if;
		axisIndex += 1;
	end_while;

END_FUNCTION

FUNCTION LMCControlCommandService::HandleRegistryCommands
	VAR_INPUT
		CommandId 	: UINT;
		Reference 	: UINT;
		pRequestFrame 	: ^USINT;
		RequestFrameSize 	: UDINT;
		pResponseFrame 	: ^USINT;
		ResponseCapacity 	: UDINT;
	END_VAR
	VAR_OUTPUT
		ResponseSize 	: DINT;
	END_VAR
	VAR
		objectNameLength : UDINT;
		objectName : ARRAY [0..255] OF CHAR;
		resolvedReference : UINT;
	END_VAR

	ResponseSize := -1;
	if (pRequestFrame = NIL) | (pResponseFrame = NIL) |
	   (RequestFrameSize < 8) then
		RETURN;
	end_if;

	case CommandId of

		0x103C:
			if ResponseCapacity < 14 then
				RETURN;
			end_if;
			resolvedReference := 0;
			if RequestFrameSize = 88 then
				(pRequestFrame + 87)^ := 0;

				if IsClientConnected(#LMCAxis1) = 1 then
					_memset(dest:=#objectName[0], usByte:=0,
						cntr:=sizeof(objectName));
					objectNameLength := _GetObjName(
						pThis:=LMCAxis1.pCmd, pName:=#objectName[0]);
					if (objectNameLength > 0) & (objectNameLength <= 79) then
						if _stricmp(str1:=(pRequestFrame + 8)$^CHAR,
							str2:=#objectName[0]) = 0 then
							resolvedReference := 1;
						end_if;
					end_if;
				end_if;

				if (resolvedReference = 0) &
				   (IsClientConnected(#LMCAxis2) = 1) then
					_memset(dest:=#objectName[0], usByte:=0,
						cntr:=sizeof(objectName));
					objectNameLength := _GetObjName(
						pThis:=LMCAxis2.pCmd, pName:=#objectName[0]);
					if (objectNameLength > 0) & (objectNameLength <= 79) then
						if _stricmp(str1:=(pRequestFrame + 8)$^CHAR,
							str2:=#objectName[0]) = 0 then
							resolvedReference := 2;
						end_if;
					end_if;
				end_if;

				if (resolvedReference = 0) &
				   (IsClientConnected(#LMCAxis3) = 1) then
					_memset(dest:=#objectName[0], usByte:=0,
						cntr:=sizeof(objectName));
					objectNameLength := _GetObjName(
						pThis:=LMCAxis3.pCmd, pName:=#objectName[0]);
					if (objectNameLength > 0) & (objectNameLength <= 79) then
						if _stricmp(str1:=(pRequestFrame + 8)$^CHAR,
							str2:=#objectName[0]) = 0 then
							resolvedReference := 3;
						end_if;
					end_if;
				end_if;

				if (resolvedReference = 0) &
				   (IsClientConnected(#LMCAxis4) = 1) then
					_memset(dest:=#objectName[0], usByte:=0,
						cntr:=sizeof(objectName));
					objectNameLength := _GetObjName(
						pThis:=LMCAxis4.pCmd, pName:=#objectName[0]);
					if (objectNameLength > 0) & (objectNameLength <= 79) then
						if _stricmp(str1:=(pRequestFrame + 8)$^CHAR,
							str2:=#objectName[0]) = 0 then
							resolvedReference := 4;
						end_if;
					end_if;
				end_if;

				if (resolvedReference = 0) &
				   (IsClientConnected(#LMCAxis5) = 1) then
					_memset(dest:=#objectName[0], usByte:=0,
						cntr:=sizeof(objectName));
					objectNameLength := _GetObjName(
						pThis:=LMCAxis5.pCmd, pName:=#objectName[0]);
					if (objectNameLength > 0) & (objectNameLength <= 79) then
						if _stricmp(str1:=(pRequestFrame + 8)$^CHAR,
							str2:=#objectName[0]) = 0 then
							resolvedReference := 5;
						end_if;
					end_if;
				end_if;

				if (resolvedReference = 0) &
				   (IsClientConnected(#LMCAxis6) = 1) then
					_memset(dest:=#objectName[0], usByte:=0,
						cntr:=sizeof(objectName));
					objectNameLength := _GetObjName(
						pThis:=LMCAxis6.pCmd, pName:=#objectName[0]);
					if (objectNameLength > 0) & (objectNameLength <= 79) then
						if _stricmp(str1:=(pRequestFrame + 8)$^CHAR,
							str2:=#objectName[0]) = 0 then
							resolvedReference := 6;
						end_if;
					end_if;
				end_if;

				if (resolvedReference = 0) &
				   (IsClientConnected(#LMCAxis7) = 1) then
					_memset(dest:=#objectName[0], usByte:=0,
						cntr:=sizeof(objectName));
					objectNameLength := _GetObjName(
						pThis:=LMCAxis7.pCmd, pName:=#objectName[0]);
					if (objectNameLength > 0) & (objectNameLength <= 79) then
						if _stricmp(str1:=(pRequestFrame + 8)$^CHAR,
							str2:=#objectName[0]) = 0 then
							resolvedReference := 7;
						end_if;
					end_if;
				end_if;

				if (resolvedReference = 0) &
				   (IsClientConnected(#LMCAxis8) = 1) then
					_memset(dest:=#objectName[0], usByte:=0,
						cntr:=sizeof(objectName));
					objectNameLength := _GetObjName(
						pThis:=LMCAxis8.pCmd, pName:=#objectName[0]);
					if (objectNameLength > 0) & (objectNameLength <= 79) then
						if _stricmp(str1:=(pRequestFrame + 8)$^CHAR,
							str2:=#objectName[0]) = 0 then
							resolvedReference := 8;
						end_if;
					end_if;
				end_if;

				if (resolvedReference = 0) &
				   (IsClientConnected(#LMCAxis9) = 1) then
					_memset(dest:=#objectName[0], usByte:=0,
						cntr:=sizeof(objectName));
					objectNameLength := _GetObjName(
						pThis:=LMCAxis9.pCmd, pName:=#objectName[0]);
					if (objectNameLength > 0) & (objectNameLength <= 79) then
						if _stricmp(str1:=(pRequestFrame + 8)$^CHAR,
							str2:=#objectName[0]) = 0 then
							resolvedReference := 9;
						end_if;
					end_if;
				end_if;
			end_if;

			if resolvedReference > 0 then
				_memset(dest:=pResponseFrame, usByte:=0, cntr:=14);
				pResponseFrame^$UINT := 0;
				(pResponseFrame + 2)^$UINT := 6;
				(pResponseFrame + 4)^$UDINT := 0;
				(pResponseFrame + 8)^$UDINT := 0;
				(pResponseFrame + 12)^$UINT := resolvedReference;
				ResponseSize := 14;
			else
				_memset(dest:=pResponseFrame, usByte:=0, cntr:=12);
				pResponseFrame^$UINT := 1;
				(pResponseFrame + 2)^$UINT := 4;
				(pResponseFrame + 4)^$UDINT := 0;
				(pResponseFrame + 8)^$UINT := 1;
				(pResponseFrame + 10)^$INT := -2;
				ResponseSize := 12;
			end_if;

		0x1042:
			if ResponseCapacity < 14 then
				RETURN;
			end_if;
			resolvedReference := 0;
			if (RequestFrameSize = 88) &
			   (IsClientConnected(#LMCRobot) = 1) then
				(pRequestFrame + 87)^ := 0;
				_memset(dest:=#objectName[0], usByte:=0,
					cntr:=sizeof(objectName));
				objectNameLength := _GetObjName(
					pThis:=LMCRobot.pCmd, pName:=#objectName[0]);
				if (objectNameLength > 0) & (objectNameLength <= 79) then
					if _stricmp(str1:=(pRequestFrame + 8)$^CHAR,
						str2:=#objectName[0]) = 0 then
						resolvedReference := 0x0100;
					end_if;
				end_if;
			end_if;

			if resolvedReference = 0x0100 then
				_memset(dest:=pResponseFrame, usByte:=0, cntr:=14);
				pResponseFrame^$UINT := 0;
				(pResponseFrame + 2)^$UINT := 6;
				(pResponseFrame + 4)^$UDINT := 0;
				(pResponseFrame + 8)^$UDINT := 0;
				(pResponseFrame + 12)^$UINT := resolvedReference;
				ResponseSize := 14;
			else
				_memset(dest:=pResponseFrame, usByte:=0, cntr:=12);
				pResponseFrame^$UINT := 1;
				(pResponseFrame + 2)^$UINT := 4;
				(pResponseFrame + 4)^$UDINT := 0;
				(pResponseFrame + 8)^$UINT := 1;
				(pResponseFrame + 10)^$INT := -2;
				ResponseSize := 12;
			end_if;

		0x202B:
			if (RequestFrameSize = 20) &
			   (Reference >= 1) & (Reference <= 9) then
				if ResponseCapacity < 16 then
					RETURN;
				end_if;
				_memset(dest:=pResponseFrame, usByte:=0, cntr:=16);
				pResponseFrame^$UINT := 0;
				(pResponseFrame + 2)^$UINT := 8;
				(pResponseFrame + 4)^$UDINT := 0;
				(pResponseFrame + 8)^$UDINT := TO_UDINT(Reference);
				(pResponseFrame + 12)^$UINT := 0;
				(pResponseFrame + 14)^$INT := 0;
				ResponseSize := 16;
			else
				if ResponseCapacity < 12 then
					RETURN;
				end_if;
				_memset(dest:=pResponseFrame, usByte:=0, cntr:=12);
				pResponseFrame^$UINT := 1;
				(pResponseFrame + 2)^$UINT := 4;
				(pResponseFrame + 4)^$UDINT := 0;
				(pResponseFrame + 8)^$UINT := 1;
				(pResponseFrame + 10)^$INT := -3;
				ResponseSize := 12;
			end_if;

	else
		ResponseSize := -1;
	end_case;

END_FUNCTION

FUNCTION LMCControlCommandService::HandleAxisCommands
	VAR_INPUT
		CommandId 	: UINT;
		Reference 	: UINT;
		pRequestFrame 	: ^USINT;
		RequestFrameSize 	: UDINT;
		pResponseFrame 	: ^USINT;
		ResponseCapacity 	: UDINT;
	END_VAR
	VAR_OUTPUT
		ResponseSize 	: DINT;
	END_VAR
	VAR
		axisCommandState : _LMCAXIS_CMDERROR;
		axisCommandStatus : UINT;
		axisCommandErrorId : INT;
		axisCommandInputValid : BOOL;
		axisClientConnected : BOOL;
		payloadReference : DINT;
		axisStatusValue : _LMCAXIS_STATUS;
		axisErrorValue : _LMCAXIS_ERROR;
		readPosition : DINT;
		position : DINT;
		speed : DINT;
		acceleration : DINT;
		deceleration : DINT;
		jerk : DINT;
		direction : DINT;
		bufferMode : DINT;
		execute : DINT;
		powerEnable : USINT;
	END_VAR

	ResponseSize := -1;
	if (pRequestFrame = NIL) | (pResponseFrame = NIL) |
	   (RequestFrameSize < 8) then
		RETURN;
	end_if;

	case CommandId of

		0x2023:
			axisCommandInputValid := FALSE;
			if RequestFrameSize = 16 then
				axisCommandInputValid :=
					(Reference >= 1) & (Reference <= 9) &
					((pRequestFrame + 8)^$UDINT = 1) &
					(((pRequestFrame + 12)^ = 0) |
					 ((pRequestFrame + 12)^ = 1)) &
					((pRequestFrame + 13)^ = 1) &
					((pRequestFrame + 14)^ = 0) &
					((pRequestFrame + 15)^ = 1);
			end_if;
			if axisCommandInputValid = FALSE then
				if ResponseCapacity < 12 then
					RETURN;
				end_if;
				_memset(dest:=pResponseFrame, usByte:=0, cntr:=12);
				pResponseFrame^$UINT := 1;
				(pResponseFrame + 2)^$UINT := 4;
				(pResponseFrame + 4)^$UDINT := 0;
				(pResponseFrame + 8)^$UINT := 1;
				(pResponseFrame + 10)^$INT := -3;
				ResponseSize := 12;
				RETURN;
			end_if;
			if ResponseCapacity < 16 then
				RETURN;
			end_if;

			powerEnable := (pRequestFrame + 12)^;
			axisCommandState := 1;
			axisClientConnected := FALSE;
			case Reference of
				1:
					if IsClientConnected(#LMCAxis1) = 1 then
						axisClientConnected := TRUE;
						OwnershipState[26] := TO_DINT(CommandId);
						OwnershipState[27] := TO_DINT(Reference);
						OwnershipState[25] := 1;
						if powerEnable = 1 then
							axisCommandState := LMCAxis1.PowerOn(
								Mode:=LMCAXIS_MOVE_SHORTEST_WAY);
						else
							axisCommandState := LMCAxis1.PowerOff(
								Mode:=LMCAXIS_SMOOTH_STOPP);
						end_if;
					end_if;
				2:
					if IsClientConnected(#LMCAxis2) = 1 then
						axisClientConnected := TRUE;
						OwnershipState[26] := TO_DINT(CommandId);
						OwnershipState[27] := TO_DINT(Reference);
						OwnershipState[25] := 1;
						if powerEnable = 1 then
							axisCommandState := LMCAxis2.PowerOn(
								Mode:=LMCAXIS_MOVE_SHORTEST_WAY);
						else
							axisCommandState := LMCAxis2.PowerOff(
								Mode:=LMCAXIS_SMOOTH_STOPP);
						end_if;
					end_if;
				3:
					if IsClientConnected(#LMCAxis3) = 1 then
						axisClientConnected := TRUE;
						OwnershipState[26] := TO_DINT(CommandId);
						OwnershipState[27] := TO_DINT(Reference);
						OwnershipState[25] := 1;
						if powerEnable = 1 then
							axisCommandState := LMCAxis3.PowerOn(
								Mode:=LMCAXIS_MOVE_SHORTEST_WAY);
						else
							axisCommandState := LMCAxis3.PowerOff(
								Mode:=LMCAXIS_SMOOTH_STOPP);
						end_if;
					end_if;
				4:
					if IsClientConnected(#LMCAxis4) = 1 then
						axisClientConnected := TRUE;
						OwnershipState[26] := TO_DINT(CommandId);
						OwnershipState[27] := TO_DINT(Reference);
						OwnershipState[25] := 1;
						if powerEnable = 1 then
							axisCommandState := LMCAxis4.PowerOn(
								Mode:=LMCAXIS_MOVE_SHORTEST_WAY);
						else
							axisCommandState := LMCAxis4.PowerOff(
								Mode:=LMCAXIS_SMOOTH_STOPP);
						end_if;
					end_if;
				5:
					if IsClientConnected(#LMCAxis5) = 1 then
						axisClientConnected := TRUE;
						OwnershipState[26] := TO_DINT(CommandId);
						OwnershipState[27] := TO_DINT(Reference);
						OwnershipState[25] := 1;
						if powerEnable = 1 then
							axisCommandState := LMCAxis5.PowerOn(
								Mode:=LMCAXIS_MOVE_SHORTEST_WAY);
						else
							axisCommandState := LMCAxis5.PowerOff(
								Mode:=LMCAXIS_SMOOTH_STOPP);
						end_if;
					end_if;
				6:
					if IsClientConnected(#LMCAxis6) = 1 then
						axisClientConnected := TRUE;
						OwnershipState[26] := TO_DINT(CommandId);
						OwnershipState[27] := TO_DINT(Reference);
						OwnershipState[25] := 1;
						if powerEnable = 1 then
							axisCommandState := LMCAxis6.PowerOn(
								Mode:=LMCAXIS_MOVE_SHORTEST_WAY);
						else
							axisCommandState := LMCAxis6.PowerOff(
								Mode:=LMCAXIS_SMOOTH_STOPP);
						end_if;
					end_if;
				7:
					if IsClientConnected(#LMCAxis7) = 1 then
						axisClientConnected := TRUE;
						OwnershipState[26] := TO_DINT(CommandId);
						OwnershipState[27] := TO_DINT(Reference);
						OwnershipState[25] := 1;
						if powerEnable = 1 then
							axisCommandState := LMCAxis7.PowerOn(
								Mode:=LMCAXIS_MOVE_SHORTEST_WAY);
						else
							axisCommandState := LMCAxis7.PowerOff(
								Mode:=LMCAXIS_SMOOTH_STOPP);
						end_if;
					end_if;
				8:
					if IsClientConnected(#LMCAxis8) = 1 then
						axisClientConnected := TRUE;
						OwnershipState[26] := TO_DINT(CommandId);
						OwnershipState[27] := TO_DINT(Reference);
						OwnershipState[25] := 1;
						if powerEnable = 1 then
							axisCommandState := LMCAxis8.PowerOn(
								Mode:=LMCAXIS_MOVE_SHORTEST_WAY);
						else
							axisCommandState := LMCAxis8.PowerOff(
								Mode:=LMCAXIS_SMOOTH_STOPP);
						end_if;
					end_if;
				9:
					if IsClientConnected(#LMCAxis9) = 1 then
						axisClientConnected := TRUE;
						OwnershipState[26] := TO_DINT(CommandId);
						OwnershipState[27] := TO_DINT(Reference);
						OwnershipState[25] := 1;
						if powerEnable = 1 then
							axisCommandState := LMCAxis9.PowerOn(
								Mode:=LMCAXIS_MOVE_SHORTEST_WAY);
						else
							axisCommandState := LMCAxis9.PowerOff(
								Mode:=LMCAXIS_SMOOTH_STOPP);
						end_if;
					end_if;
			else
			end_case;
			if axisClientConnected = TRUE then
				axisCommandStatus := axisCommandState$UINT;
				axisCommandErrorId := axisCommandState$INT;
				if (axisCommandState$UDINT and 0xFFFF0000) <> 0 then
					axisCommandStatus := 1;
					axisCommandErrorId := -6;
				end_if;
			else
				axisCommandStatus := 1;
				axisCommandErrorId := -2;
			end_if;
			_memset(dest:=pResponseFrame, usByte:=0, cntr:=16);
			pResponseFrame^$UINT := 0;
			(pResponseFrame + 2)^$UINT := 8;
			(pResponseFrame + 4)^$UDINT := 0;
			(pResponseFrame + 8)^$UDINT := TO_UDINT(Reference);
			(pResponseFrame + 12)^$UINT := axisCommandStatus;
			(pResponseFrame + 14)^$INT := axisCommandErrorId;
			ResponseSize := 16;

		0x2024:
			axisCommandInputValid := FALSE;
			if RequestFrameSize = 9 then
				axisCommandInputValid :=
					((pRequestFrame + 8)^ = 1) &
					(Reference >= 1) & (Reference <= 9);
			end_if;
			if axisCommandInputValid = FALSE then
				if ResponseCapacity < 12 then
					RETURN;
				end_if;
				_memset(dest:=pResponseFrame, usByte:=0, cntr:=12);
				pResponseFrame^$UINT := 1;
				(pResponseFrame + 2)^$UINT := 4;
				(pResponseFrame + 4)^$UDINT := 0;
				(pResponseFrame + 8)^$UINT := 1;
				(pResponseFrame + 10)^$INT := -3;
				ResponseSize := 12;
				RETURN;
			end_if;
			if ResponseCapacity < 16 then
				RETURN;
			end_if;
			axisCommandStatus := 1;
			axisCommandErrorId := -2;
			axisClientConnected := FALSE;
			case Reference of
				1:
					if IsClientConnected(#LMCAxis1) = 1 then
						axisClientConnected := TRUE;
						OwnershipState[26] := TO_DINT(CommandId);
						OwnershipState[27] := TO_DINT(Reference);
						OwnershipState[25] := 1;
						LMCAxis1.QuitError();
					end_if;
				2:
					if IsClientConnected(#LMCAxis2) = 1 then
						axisClientConnected := TRUE;
						OwnershipState[26] := TO_DINT(CommandId);
						OwnershipState[27] := TO_DINT(Reference);
						OwnershipState[25] := 1;
						LMCAxis2.QuitError();
					end_if;
				3:
					if IsClientConnected(#LMCAxis3) = 1 then
						axisClientConnected := TRUE;
						OwnershipState[26] := TO_DINT(CommandId);
						OwnershipState[27] := TO_DINT(Reference);
						OwnershipState[25] := 1;
						LMCAxis3.QuitError();
					end_if;
				4:
					if IsClientConnected(#LMCAxis4) = 1 then
						axisClientConnected := TRUE;
						OwnershipState[26] := TO_DINT(CommandId);
						OwnershipState[27] := TO_DINT(Reference);
						OwnershipState[25] := 1;
						LMCAxis4.QuitError();
					end_if;
				5:
					if IsClientConnected(#LMCAxis5) = 1 then
						axisClientConnected := TRUE;
						OwnershipState[26] := TO_DINT(CommandId);
						OwnershipState[27] := TO_DINT(Reference);
						OwnershipState[25] := 1;
						LMCAxis5.QuitError();
					end_if;
				6:
					if IsClientConnected(#LMCAxis6) = 1 then
						axisClientConnected := TRUE;
						OwnershipState[26] := TO_DINT(CommandId);
						OwnershipState[27] := TO_DINT(Reference);
						OwnershipState[25] := 1;
						LMCAxis6.QuitError();
					end_if;
				7:
					if IsClientConnected(#LMCAxis7) = 1 then
						axisClientConnected := TRUE;
						OwnershipState[26] := TO_DINT(CommandId);
						OwnershipState[27] := TO_DINT(Reference);
						OwnershipState[25] := 1;
						LMCAxis7.QuitError();
					end_if;
				8:
					if IsClientConnected(#LMCAxis8) = 1 then
						axisClientConnected := TRUE;
						OwnershipState[26] := TO_DINT(CommandId);
						OwnershipState[27] := TO_DINT(Reference);
						OwnershipState[25] := 1;
						LMCAxis8.QuitError();
					end_if;
				9:
					if IsClientConnected(#LMCAxis9) = 1 then
						axisClientConnected := TRUE;
						OwnershipState[26] := TO_DINT(CommandId);
						OwnershipState[27] := TO_DINT(Reference);
						OwnershipState[25] := 1;
						LMCAxis9.QuitError();
					end_if;
			else
			end_case;
			if axisClientConnected = TRUE then
				axisCommandStatus := 0;
				axisCommandErrorId := 0;
			end_if;
			_memset(dest:=pResponseFrame, usByte:=0, cntr:=16);
			pResponseFrame^$UINT := 0;
			(pResponseFrame + 2)^$UINT := 8;
			(pResponseFrame + 4)^$UDINT := 0;
			(pResponseFrame + 8)^$UDINT := TO_UDINT(Reference);
			(pResponseFrame + 12)^$UINT := axisCommandStatus;
			(pResponseFrame + 14)^$INT := axisCommandErrorId;
			ResponseSize := 16;

		0x2022:
			if (RequestFrameSize <> 24) |
			   (Reference < 1) | (Reference > 9) then
				if ResponseCapacity < 12 then
					RETURN;
				end_if;
				_memset(dest:=pResponseFrame, usByte:=0, cntr:=12);
				pResponseFrame^$UINT := 1;
				(pResponseFrame + 2)^$UINT := 4;
				(pResponseFrame + 4)^$UDINT := 0;
				(pResponseFrame + 8)^$UINT := 1;
				(pResponseFrame + 10)^$INT := -3;
				ResponseSize := 12;
				RETURN;
			end_if;
			if ResponseCapacity < 16 then
				RETURN;
			end_if;
			deceleration := (pRequestFrame + 8)^$DINT;
			jerk := (pRequestFrame + 12)^$DINT;
			bufferMode := (pRequestFrame + 16)^$DINT;
			execute := (pRequestFrame + 20)^$DINT;
			axisCommandInputValid := (bufferMode = 1) & (execute = 1) &
				(deceleration > 0) & (jerk >= 0);
			axisCommandState := 1;
			axisClientConnected := FALSE;
			if axisCommandInputValid = TRUE then
				case Reference of
					1:
						if IsClientConnected(#LMCAxis1) = 1 then
							axisClientConnected := TRUE;
							OwnershipState[26] := TO_DINT(CommandId);
							OwnershipState[27] := TO_DINT(Reference);
							OwnershipState[25] := 1;
							axisCommandState := LMCAxis1.StopMove(
								Decel:=deceleration, Jerk:=jerk);
						end_if;
					2:
						if IsClientConnected(#LMCAxis2) = 1 then
							axisClientConnected := TRUE;
							OwnershipState[26] := TO_DINT(CommandId);
							OwnershipState[27] := TO_DINT(Reference);
							OwnershipState[25] := 1;
							axisCommandState := LMCAxis2.StopMove(
								Decel:=deceleration, Jerk:=jerk);
						end_if;
					3:
						if IsClientConnected(#LMCAxis3) = 1 then
							axisClientConnected := TRUE;
							OwnershipState[26] := TO_DINT(CommandId);
							OwnershipState[27] := TO_DINT(Reference);
							OwnershipState[25] := 1;
							axisCommandState := LMCAxis3.StopMove(
								Decel:=deceleration, Jerk:=jerk);
						end_if;
					4:
						if IsClientConnected(#LMCAxis4) = 1 then
							axisClientConnected := TRUE;
							OwnershipState[26] := TO_DINT(CommandId);
							OwnershipState[27] := TO_DINT(Reference);
							OwnershipState[25] := 1;
							axisCommandState := LMCAxis4.StopMove(
								Decel:=deceleration, Jerk:=jerk);
						end_if;
					5:
						if IsClientConnected(#LMCAxis5) = 1 then
							axisClientConnected := TRUE;
							OwnershipState[26] := TO_DINT(CommandId);
							OwnershipState[27] := TO_DINT(Reference);
							OwnershipState[25] := 1;
							axisCommandState := LMCAxis5.StopMove(
								Decel:=deceleration, Jerk:=jerk);
						end_if;
					6:
						if IsClientConnected(#LMCAxis6) = 1 then
							axisClientConnected := TRUE;
							OwnershipState[26] := TO_DINT(CommandId);
							OwnershipState[27] := TO_DINT(Reference);
							OwnershipState[25] := 1;
							axisCommandState := LMCAxis6.StopMove(
								Decel:=deceleration, Jerk:=jerk);
						end_if;
					7:
						if IsClientConnected(#LMCAxis7) = 1 then
							axisClientConnected := TRUE;
							OwnershipState[26] := TO_DINT(CommandId);
							OwnershipState[27] := TO_DINT(Reference);
							OwnershipState[25] := 1;
							axisCommandState := LMCAxis7.StopMove(
								Decel:=deceleration, Jerk:=jerk);
						end_if;
					8:
						if IsClientConnected(#LMCAxis8) = 1 then
							axisClientConnected := TRUE;
							OwnershipState[26] := TO_DINT(CommandId);
							OwnershipState[27] := TO_DINT(Reference);
							OwnershipState[25] := 1;
							axisCommandState := LMCAxis8.StopMove(
								Decel:=deceleration, Jerk:=jerk);
						end_if;
					9:
						if IsClientConnected(#LMCAxis9) = 1 then
							axisClientConnected := TRUE;
							OwnershipState[26] := TO_DINT(CommandId);
							OwnershipState[27] := TO_DINT(Reference);
							OwnershipState[25] := 1;
							axisCommandState := LMCAxis9.StopMove(
								Decel:=deceleration, Jerk:=jerk);
						end_if;
				else
				end_case;
			end_if;
			if axisClientConnected = TRUE then
				axisCommandStatus := axisCommandState$UINT;
				axisCommandErrorId := axisCommandState$INT;
				if (axisCommandState$UDINT and 0xFFFF0000) <> 0 then
					axisCommandStatus := 1;
					axisCommandErrorId := -6;
				end_if;
			elsif axisCommandInputValid = TRUE then
				axisCommandStatus := 1;
				axisCommandErrorId := -2;
			else
				axisCommandStatus := 1;
				axisCommandErrorId := -7;
			end_if;
			_memset(dest:=pResponseFrame, usByte:=0, cntr:=16);
			pResponseFrame^$UINT := 0;
			(pResponseFrame + 2)^$UINT := 8;
			(pResponseFrame + 4)^$UDINT := 0;
			(pResponseFrame + 8)^$UDINT := TO_UDINT(Reference);
			(pResponseFrame + 12)^$UINT := axisCommandStatus;
			(pResponseFrame + 14)^$INT := axisCommandErrorId;
			ResponseSize := 16;

		0x2028:
			axisCommandErrorId := -3;
			axisCommandStatus := 1;
			axisStatusValue := 0;
			axisErrorValue := 0;
			payloadReference := 0;
			execute := 0;
			if RequestFrameSize >= 16 then
				payloadReference := (pRequestFrame + 8)^$DINT;
				execute := (pRequestFrame + 12)^$DINT;
			end_if;
			if (RequestFrameSize = 16) &
			   (Reference >= 1) & (Reference <= 9) &
			   (payloadReference = TO_DINT(Reference)) & (execute = 1) then
				if ResponseCapacity < 20 then
					RETURN;
				end_if;
				axisCommandErrorId := -2;
				case Reference of
					1:
						if IsClientConnected(#LMCAxis1) = 1 then
							axisStatusValue := LMCAxis1.ReadAxisStatus();
							axisErrorValue := LMCAxis1.ReadAxisError();
							axisCommandStatus := 0;
							axisCommandErrorId := 0;
						end_if;
					2:
						if IsClientConnected(#LMCAxis2) = 1 then
							axisStatusValue := LMCAxis2.ReadAxisStatus();
							axisErrorValue := LMCAxis2.ReadAxisError();
							axisCommandStatus := 0;
							axisCommandErrorId := 0;
						end_if;
					3:
						if IsClientConnected(#LMCAxis3) = 1 then
							axisStatusValue := LMCAxis3.ReadAxisStatus();
							axisErrorValue := LMCAxis3.ReadAxisError();
							axisCommandStatus := 0;
							axisCommandErrorId := 0;
						end_if;
					4:
						if IsClientConnected(#LMCAxis4) = 1 then
							axisStatusValue := LMCAxis4.ReadAxisStatus();
							axisErrorValue := LMCAxis4.ReadAxisError();
							axisCommandStatus := 0;
							axisCommandErrorId := 0;
						end_if;
					5:
						if IsClientConnected(#LMCAxis5) = 1 then
							axisStatusValue := LMCAxis5.ReadAxisStatus();
							axisErrorValue := LMCAxis5.ReadAxisError();
							axisCommandStatus := 0;
							axisCommandErrorId := 0;
						end_if;
					6:
						if IsClientConnected(#LMCAxis6) = 1 then
							axisStatusValue := LMCAxis6.ReadAxisStatus();
							axisErrorValue := LMCAxis6.ReadAxisError();
							axisCommandStatus := 0;
							axisCommandErrorId := 0;
						end_if;
					7:
						if IsClientConnected(#LMCAxis7) = 1 then
							axisStatusValue := LMCAxis7.ReadAxisStatus();
							axisErrorValue := LMCAxis7.ReadAxisError();
							axisCommandStatus := 0;
							axisCommandErrorId := 0;
						end_if;
					8:
						if IsClientConnected(#LMCAxis8) = 1 then
							axisStatusValue := LMCAxis8.ReadAxisStatus();
							axisErrorValue := LMCAxis8.ReadAxisError();
							axisCommandStatus := 0;
							axisCommandErrorId := 0;
						end_if;
					9:
						if IsClientConnected(#LMCAxis9) = 1 then
							axisStatusValue := LMCAxis9.ReadAxisStatus();
							axisErrorValue := LMCAxis9.ReadAxisError();
							axisCommandStatus := 0;
							axisCommandErrorId := 0;
						end_if;
				else
				end_case;
				_memset(dest:=pResponseFrame, usByte:=0, cntr:=20);
				pResponseFrame^$UINT := 0;
				(pResponseFrame + 2)^$UINT := 12;
				(pResponseFrame + 4)^$UDINT := 0;
				(pResponseFrame + 8)^$UDINT := axisStatusValue$UDINT;
				(pResponseFrame + 12)^$UINT := axisCommandStatus;
				(pResponseFrame + 14)^$INT := axisCommandErrorId;
				(pResponseFrame + 16)^$UINT := axisErrorValue$UINT;
				(pResponseFrame + 18)^$UINT := 0;
				ResponseSize := 20;
			else
				if ResponseCapacity < 12 then
					RETURN;
				end_if;
				_memset(dest:=pResponseFrame, usByte:=0, cntr:=12);
				pResponseFrame^$UINT := 1;
				(pResponseFrame + 2)^$UINT := 4;
				(pResponseFrame + 4)^$UDINT := 0;
				(pResponseFrame + 8)^$UINT := 1;
				(pResponseFrame + 10)^$INT := axisCommandErrorId;
				ResponseSize := 12;
			end_if;
